// TwinCAT 3 PLC project PLC_PML
// ProgramVersion: 3.1.4023.0
// libraries:
//   Tc2_MC2, * (Beckhoff Automation GmbH)
//   Tc2_MC2_Drive, * (Beckhoff Automation GmbH)
//   Tc2_Standard, * (Beckhoff Automation GmbH)
//   Tc2_System, * (Beckhoff Automation GmbH)
//   Tc3_EventLogger, * (Beckhoff Automation GmbH)
//   Tc3_Module, * (Beckhoff Automation GmbH)
//   Tc3_PackML_V2, * (Beckhoff Automation GmbH)
// project tree:
//   Application/01_Application_Level_Items/02_DUT/01_ENUM/ E_PMLUnitMode.TcDUT
//   Application/01_Application_Level_Items/02_DUT/03_ALIAS/ T_PackMLTags.TcDUT
//   Application/01_Application_Level_Items/99_VISU/ V_Application.TcVIS
//   Application/02_MachineModules/ FB_TestMachine.TcPOU
//   Application/03_EquipmentModules/ FB_TestEquipment.TcPOU
//   Application/04_ControlModules/ FB_TestControl.TcPOU
//   Application/ MAIN.TcPOU
//   Base/01_PML/01_Module/01_Base/02_DUT/ ST_PMLModuleBase_HMI.TcDUT, ST_PMLModuleBase_VISU.TcDUT, ST_PMLSubUnitInfoExt.TcDUT
//   Base/01_PML/01_Module/01_Base/03_ITFs/ ITF_PMLModuleBase.TcIO
//   Base/01_PML/01_Module/01_Base/ FB_PMLModuleBase.TcPOU
//   Base/01_PML/01_Module/02_Events/ FB_PMLModeLogger.TcPOU, FB_PMLStateLogger.TcPOU
//   Base/01_PML/01_Module/03_PMLControl/03_ITFs/ ITF_PackML_ExternalControl.TcIO, ITF_PackML_ExternalControl_Simplified.TcIO
//   Base/01_PML/01_Module/03_PMLControl/ FB_ModuleExternalCommandControl.TcPOU, FB_PackML_ExternalControl.TcPOU, FB_PackML_PushButtonControl.TcPOU, ITF_PackML_ExternalControl_Simplified_old.TcIO
//   Base/01_PML/01_Module/04_SequenceControl/ E_ModuleSequenceCommand.TcDUT, E_ModuleSequenceStatus.TcDUT, F_CommandAllSequences.TcPOU, ITF_ModuleSequenceControl.TcIO, ST_ModuleSequenceControl.TcDUT
//   Base/01_PML/01_Module/05_Visualizations/ V_Module.TcVIS
//   Base/01_PML/02_GVL/ GVL_PML_Base.TcGVL
//   Base/01_PML/03_Visualizations/ V_MachineModule.TcVIS
//   Base/01_PML/99_Templates/01_ModuleTemplate/ FB_ApplicationModule_TEMPLATE.TcPOU
//   Base/02_Components/01_Base/ FB_ComponentBase.TcPOU, ITF_ComponentBase.TcIO, ST_ComponentBase_HMI.TcDUT
//   Base/02_Components/02_Axes/01_Base/ FB_AxisBase.TcPOU, ITF_AxisBase.TcIO, ST_AxisBase_HMI.TcDUT
//   Base/02_Components/02_Axes/02_Homing/ FB_Axis_HomeToSensor.TcPOU, FB_Axis_NoHoming.TcPOU
//   Base/02_Components/02_Axes/03_MotionType/ FB_Axis_Continuous_HomeToSensor.TcPOU, FB_Axis_Continuous_NoHoming.TcPOU, FB_Axis_Discrete_HomeToSensor.TcPOU, ITF_Axis_Continuous.TcIO, ITF_Axis_Discrete.TcIO
//   Base/02_Components/03_Cylinders/01_Base/ FB_CylinderBase.TcPOU, ITF_CylinderBase.TcIO, ST_CylinderBase_HMI.TcDUT
//   Base/02_Components/03_Cylinders/02_Feedback/ FB_Cylinder_DualSensor.TcPOU
//   Base/02_Components/03_Cylinders/03_Actuation/ FB_Cylinder_DualSolenoid_DualSensor.TcPOU
//   Base/02_Components/04_Sensors/01_Base/ E_DebounceMode.TcDUT, E_SensorSimulationMode.TcDUT, FB_SensorBase.TcPOU, ITF_SensorBase.TcIO, ST_SensorBase_HMI.TcDUT
//   Base/02_Components/04_Sensors/02_Sensor/ FB_Sensor.TcPOU
//   Base/03_Utilities/01_Events/ F_CreateAllEventsInClass.TcPOU
//   Base/03_Utilities/02_DataStructures/01_Tree/01_Tree_IndexBased/ FB_Tree_IndexBased.TcPOU, ITF_Tree_IndexBased.TcIO, ST_Tree_IndexBased_Node.TcDUT
//   Base/03_Utilities/03_HMI_Connections/ FB_MainHMI_Connection.TcPOU
//   / GlobalTextList.TcGTLO, PlcTask.TcTTO, Visualization Manager.TcVMO (not stored)
// real-time tasks:
//   TASK PlcTask: cycle T#1ms, priority 20, ADS port 350
//   TASK VISU_TASK: cycle T#200000us, priority 30, ADS port 351
//   TASK Job Task: cycle default, priority 32
//   TASK MC-Task (MET): cycle T#2ms, priority 3, ADS port 521
//   TASK MC-Task (MPT): cycle T#10ms, priority 8, ADS port 531
// motion (NC):
//   TASK NC-Task 1 SAF: cycle T#2ms, priority 4, ADS port 501
//   TASK NC-Task 1 SVB: cycle T#10ms, priority 9, ADS port 511
//   AXIS Axis 1 (id 1)
//     General: UnitFlags=#x00000004
//     Dynamic: AccelerationMaximum=10000, DecelerationMaximum=10000, Acceleration=1000, Deceleration=1000, Jerk=1750
//     Velo: Maximum=1500
//     OtherSettings: AllowMotionCmdToSlave=true
//     encoder EncType=1
//       EncPara: ModuloFactor=720
//     drive DrvType=5
//       Analog: TorqueSetpointScale=10, ScaleFactorActTorque=0.1
//       TimeComp: TaskDelayCycles=1
//     controller CtrType=1
//       CtrPara: PriorControlFactor=1
//         Observer: BandWidth=20
//   AXIS Axis 2 (id 2)
//     General: UnitFlags=#x00000004
//     OtherSettings: AllowMotionCmdToSlave=true
//     encoder EncType=1
//     drive DrvType=5
//       Analog: TorqueSetpointScale=10, ScaleFactorActTorque=0.1
//       TimeComp: TaskDelayCycles=1
//     controller CtrType=1
//       CtrPara: PriorControlFactor=1
//         Observer: BandWidth=20
// variable links:
//   PLC_PML/PLC_PML Instance <-> NC-Task 1 SAF/Axes/Axis 1
//     PlcTask Inputs/MAIN.fbMyMachine.fbEquipmentModule1.fb_EM1_ControlModule1.fbAxis1.HardwareAxis.NcToPlc <-> Outputs/ToPlc
//     PlcTask Outputs/MAIN.fbMyMachine.fbEquipmentModule1.fb_EM1_ControlModule1.fbAxis1.HardwareAxis.PlcToNc <-> Inputs/FromPlc
//   PLC_PML/PLC_PML Instance <-> NC-Task 1 SAF/Axes/Axis 2
//     PlcTask Inputs/MAIN.fbMyMachine.fbEquipmentModule1.fb_EM1_ControlModule1.fbAxis1.SimulationAxis.NcToPlc <-> Outputs/ToPlc
//     PlcTask Outputs/MAIN.fbMyMachine.fbEquipmentModule1.fb_EM1_ControlModule1.fbAxis1.SimulationAxis.PlcToNc <-> Inputs/FromPlc

CONFIGURATION PLC_PML
    RESOURCE PLC ON TwinCAT3
        TASK PlcTask(INTERVAL := T#1ms, PRIORITY := 20);
        PROGRAM MAIN WITH PlcTask : MAIN;
    END_RESOURCE
END_CONFIGURATION

// ---- Application/01_Application_Level_Items/02_DUT/01_ENUM/E_PMLUnitMode.TcDUT
{attribute 'qualified_only'}		//Note that this is not "Strict" since it needs to interact with the mode manager, which uses DINTs for mode
TYPE E_PMLUnitMode:
(
	ePMLUnitMode_Invalid 		:= 0,
	ePMLUnitMode_Production		:= 1,
	ePMLUnitMode_Maintenance	:= 2,
	ePMLUnitMode_Manual			:= 3
	// User defined modes
    (*ePMLUnitMode_SemiAutomatic  :=  4,
    ePMLUnitMode_DryRun         :=  5,
	ePMLUnitMode_Standalone		:=  6,
	ePMLUnitMode_Usermode4		:=  7,
	ePMLUnitMode_Usermode5 		:=  8,
	ePMLUnitMode_Usermode6 		:=  9,
	ePMLUnitMode_Usermode7 		:=  10 *)	
) DINT;
END_TYPE

// ---- Application/01_Application_Level_Items/02_DUT/03_ALIAS/T_PackMLTags.TcDUT
(*	Change the type depending on the needs, minimum packml set or full
Tc3_PackML_V2.ST_PackMLv30 // Tc3_PackML_V2.ST_PackMLv30min*)
TYPE T_PackMLTags : Tc3_PackML_V2.ST_PackMLv30; END_TYPE

// ---- Base/01_PML/01_Module/01_Base/02_DUT/ST_PMLModuleBase_HMI.TcDUT
TYPE ST_PMLModuleBase_HMI :
STRUCT
	bEnabled			: BOOL;					//Enables or disables the packml Machine of the module (prevents the module from going past idle)
	eMode				: E_PMLUnitMode;		//Current UnitMode of the module
	nModuleID			: DINT;					//Unique identifying number for the module
	sModuleName			: STRING;				//Human-readable module name for user-side messaging
	eState				: Tc3_PackML_V2.E_PMLState;
	bLogStateChanges 	: BOOL := TRUE; 		//Toggle to permit or suppress state change logging (Should be tied to HMI setting to optionally reduce event logger clutter)
	bLogModeChanges 	: BOOL := TRUE; 		//Toggle to permit or suppress state change logging (Should be tied to HMI setting to optionally reduce event logger clutter)
	
	//Control information
	bHMIControlAvailable	: BOOL;		//Set TRUE *FROM PLC* when HMI requests can be processed
	bIncomingHMIRequest 	: BOOL;		//Pulses TRUE when an HMI request is issued
	bHMICommandConfirmation	: BOOL;		//Confirms receipt and subsequent processing of the command sent by the HMI
	
	bModeCommandHMIRequest	: BOOL;		//Pulses TRUE when an HMI mode change request is issued
	bStateCommandHMIRequest	: BOOL;		//Pulses TRUE when an HMI state change request is issued
	bEnableHMIRequest				: BOOL;		//HMI requests to enable the module
	bDisableHMIRequest 				: BOOL;		//HMI requests to disable the module
	bActivateStateLogHMIRequest			: BOOL;		//HMI requests to enable the module
	bDeactivateStateLogHMIRequest 		: BOOL;		//HMI requests to disable the module
	bActivateModeLogHMIRequest			: BOOL;		//HMI requests to enable the module
	bDeactivateModeLogHMIRequest 		: BOOL;		//HMI requests to disable the module
	eModeCommandHMIValue			: E_PMLUnitMode;
	eStateCommandHMIValue			: Tc3_PackML_V2.E_PMLCommand;
	
END_STRUCT
END_TYPE

// ---- Base/01_PML/01_Module/01_Base/02_DUT/ST_PMLModuleBase_VISU.TcDUT
TYPE ST_PMLModuleBase_VISU :
STRUCT
	bEnabled			: BOOL;					//Enables or disables the packml Machine of the module (prevents the module from going past idle)
	eMode				: E_PMLUnitMode;		//Current UnitMode of the module
	nModuleID			: DINT;					//Unique identifying number for the module
	sModuleName			: STRING;				//Human-readable module name for user-side messaging
	eState				: Tc3_PackML_V2.E_PMLState;
	
	//eModeCommandValue	: E_PMLUnitMode;
	///eStateCommandValue	: Tc3_PackML_V2.E_PMLCommand;
	bStartPressed		: BOOL;
	///bStartEnabled		: BOOL;
	bStopPressed		: BOOL;
	///bStopEnabled		: BOOL;
	bResetPressed		: BOOL;
	///bResetEnabled		: BOOL;
	bClearPressed		: BOOL;
	///bClearEnabled		: BOOL;	
	
	bAbortPressed		: BOOL;
	bHoldPressed		: BOOL;
	bUnholdPressed		: BOOL;
	bSuspendPressed		: BOOL;
	bUnsuspendPressed	: BOOL;
	
	// Mode things
	bProductionPressed	: BOOL;
	bMaintenancePressed	: BOOL;
	bManualPressed		: BOOL;
	
END_STRUCT
END_TYPE

// ---- Base/01_PML/01_Module/01_Base/02_DUT/ST_PMLSubUnitInfoExt.TcDUT
TYPE ST_PMLSubUnitInfoExt EXTENDS ST_PMLSubUnitInfo :	//Extended Struct of ST_PMLSubUnitInfo
STRUCT
	nModuleID 						: DINT; 				//Machine ID for messaging and Identification
	sModuleName						: STRING;				//Human readable machine name for messaging
	UnitModeCurrent					: E_PMLProtectedUnitMode;
	ActiveAlarm						: BOOL;
END_STRUCT
END_TYPE

// ---- Base/01_PML/01_Module/04_SequenceControl/E_ModuleSequenceCommand.TcDUT
{attribute 'qualified_only'}
{attribute 'strict'}
TYPE E_ModuleSequenceCommand :
(
	Enable,
	Disable,
	Start,
	Resume,
	Reset,
	Clear	
);
END_TYPE

// ---- Base/01_PML/01_Module/04_SequenceControl/E_ModuleSequenceStatus.TcDUT
{attribute 'qualified_only'}
{attribute 'strict'}
TYPE E_ModuleSequenceStatus :
(
	Idle,
	Busy,
	Waiting,
	Complete,
	Disabled,
	Error
);
END_TYPE

// ---- Base/01_PML/01_Module/04_SequenceControl/ST_ModuleSequenceControl.TcDUT
TYPE ST_ModuleSequenceControl :
STRUCT
	eCommand				: E_ModuleSequenceCommand;	//Command Enumeration
	bNewCommand				: BOOL;						//Pulses TRUE when a new command is received
	bSequenceStateChange	: BOOL;						//TRUE when the sequence is transitioning between states, allows for one shot "on entry" tasks in sequence states 
	eStatus					: E_ModuleSequenceStatus;	//Abstracted and generalized status information for the local state machine status
END_STRUCT
END_TYPE

// ---- Base/02_Components/01_Base/ST_ComponentBase_HMI.TcDUT
TYPE ST_ComponentBase_HMI :
STRUCT
	//Status information
	bEnabled	: BOOL;
	bSimulate 	: BOOL;
	sName		: STRING;
	bActive		: BOOL;
	bError		: BOOL;
	nErrorID	: UDINT;
	
	//Control information
	bHMIControlAvailable	: BOOL;		//Set TRUE *FROM PLC* when HMI requests can be processed
	bIncomingHMIRequest 	: BOOL;		//Pulses TRUE when an HMI request is issued
	bHMICommandConfirmation	: BOOL;		//Confirms receipt and subsequent processing of the command sent by the HMI
	
	bEnableHMIRequest				: BOOL;		//HMI requests to enable the component
	bDisableHMIRequest 				: BOOL;		//HMI requests to disable the component
	bSimulateOperationHMIRequest 	: BOOL;		//HMI requests to change the component to simulation mode
	bStandardOperationHMIRequest	: BOOL;		//HMI requests to change the component to standard mode
	bResetHMIRequest				: BOOL;		//HMI requests to reset the component
	
END_STRUCT
END_TYPE

// ---- Base/02_Components/02_Axes/01_Base/ST_AxisBase_HMI.TcDUT
TYPE ST_AxisBase_HMI :
STRUCT
	fJogFastVelocity	: LREAL;
	fJogSlowVelocity	: LREAL;
	fTargetVelocity		: LREAL;
	
	bDriveEnabled		: BOOL;
	bInGear				: BOOL;
	bInPosition			: BOOL;
	fPosition 			: LREAL;
	fPositionSetpoint	: LREAL;
	bStopped			: BOOL;
	
	//Control information
	bHMIControlAvailable	: BOOL;		//Set TRUE *FROM PLC* when HMI requests can be processed
	bIncomingHMIRequest 	: BOOL;		//Pulses TRUE when an HMI request is issued
		bHMICommandConfirmation	: BOOL;		//Confirms receipt and subsequent processing of the command sent by the HMI
	
	bDriveEnableHMIRequest				: BOOL;		//HMI requests to enable the axis
	bDriveDisableHMIRequest 				: BOOL;		//HMI requests to disable the axis
	bSetJogFastVelocityRequest		: BOOL;
	bSetJogSlowVelocityRequest		: BOOL;
	fSetJogFastVelocityValue		: LREAL;
	fSetJogSlowVelocityValue		: LREAL;
	bSetTargetVelocityRequest		: BOOL;
	bSetTargetVelocityValue			: LREAL;
END_STRUCT
END_TYPE

// ---- Base/02_Components/03_Cylinders/01_Base/ST_CylinderBase_HMI.TcDUT
TYPE ST_CylinderBase_HMI:
STRUCT
	//Status information
	tExtendTime		: TIME;
	tRetractTime	: TIME;
	fTimeoutFactor	: LREAL;
	bExtended		: BOOL;
	bRetracted		: BOOL;
	bExtending		: BOOL;
	bRetracting		: BOOL;
	bRetractCommand	: BOOL;
	bExtendCommand	: BOOL;
	
	//Control information
	bHMIControlAvailable	: BOOL;		//Set TRUE *FROM PLC* when HMI requests can be processed
	bIncomingHMIRequest 	: BOOL;		//Pulses TRUE when an HMI request is issued
		bHMICommandConfirmation	: BOOL;		//Confirms receipt and subsequent processing of the command sent by the HMI
	
	bExtendHMIRequest			: BOOL;			//HMI requests to extend the cylinder
	bRetractHMIRequest			: BOOL;			//HMI requests to retract the cylinder
	bIdleHMIRequest				: BOOL;			//HMI requests to idle the cylinder (no active output)
	bExtendTimeHMISetRequest	: BOOL;			//HMI requests to set the cylinder's expected extend time
	tExtendTimeHMISetValue		: TIME;			//HMI setpoint value for the expected extend time
	bRetractTimeHMISetRequest	: BOOL;			//HMI requests to set the cylinder's expected retract time
	tRetractTimeHMISetValue		: TIME;			//HMI setpoint value for the expected retract time
	bTimeoutFactorHMISetRequest	: BOOL;			//HMI requests to set the timeout factor for the cylinder
	fTimeoutFactorHMISetValue	: LREAL;		//HMI setpoint value for the cylinder's timeout factor
END_STRUCT
END_TYPE

// ---- Base/02_Components/04_Sensors/01_Base/E_DebounceMode.TcDUT
{attribute 'qualified_only'}
{attribute 'strict'}
TYPE E_DebounceMode :
(
	RawInput,
	SimpleFlickerFilter,
	EdgeDetectFilter,
	MovingAverage
) DINT;
END_TYPE

// ---- Base/02_Components/04_Sensors/01_Base/E_SensorSimulationMode.TcDUT
{attribute 'qualified_only'}
{attribute 'strict'}
TYPE E_SensorSimulationMode :
(
	InputDriven,		//Follows the state of the SimulationInput property
	Periodic			//Follows a 50% duty cycle at the period specified in ms by SimulationInput);
);
END_TYPE

// ---- Base/02_Components/04_Sensors/01_Base/ST_SensorBase_HMI.TcDUT
TYPE ST_SensorBase_HMI :
STRUCT
	//Status information
	eDebounceMode		: E_DebounceMode;
	tDebounceTime 		: TIME;
	bInverted			: BOOL;
	eSimulationMode		: E_SensorSimulationMode;
	nSimulationInput	: DINT;
	tTimeActive			: TIME;
	tTimeInactive		: TIME;
	
	//Control information
	bHMIControlAvailable	: BOOL;		//Set TRUE *FROM PLC* when HMI requests can be processed
	bIncomingHMIRequest 	: BOOL;		//Pulses TRUE when an HMI request is issued
		bHMICommandConfirmation	: BOOL;		//Confirms receipt and subsequent processing of the command sent by the HMI
	
	bSetDebounceModeHMIRequest 		: BOOL;		//HMI requests to change the Debounce mode of the sensor
	eSetDebounceModeHMIValue 		: E_DebounceMode;			//HMI requested Debounce mode of the sensor
	bSetDebounceTimeHMIRequest		: BOOL;		//HMI requests to change the Debounce time of the sensor
	tSetDebounceTimeHMIValue 		: TIME;	//HMI requested Debounce mode of the sensor
	bSetSimulationModeHMIRequest	: BOOL;		//HMI requests to change the simulation mode of the sensor
	eSetSimulationModeHMIValue		: E_SensorSimulationMode;	//HMI Requested Simulation mode of the sensor
	bSetSimulationInputHMIRequest	: BOOL;		//HMI requests to set the simulation input value
	nSetSimulationInputHMIValue		: DINT;		//HMI requested simulation input value
	bInvertedHMIRequest				: BOOL;		//HMI requests that the sensor operate in an inverted state
	bUninvertedHMIRequest			: BOOL;		//HMI requests that the sensor operate in an uninverted state
	
	bSimulateOperationHMIRequest 	: BOOL;		//HMI requests to change the component to simulation mode
	bStandardOperationHMIRequest	: BOOL;		//HMI requests to change the component to standard mode

END_STRUCT
END_TYPE

// ---- Base/03_Utilities/02_DataStructures/01_Tree/01_Tree_IndexBased/ST_Tree_IndexBased_Node.TcDUT
TYPE ST_Tree_IndexBased_Node :
STRUCT
	sName 		: STRING;
	nChildCount	: DINT;
	nParent		: DINT;
	a_nChildren	: ARRAY[0..15] OF DINT;
	nDepth		: DINT;
END_STRUCT
END_TYPE

// ---- Base/01_PML/02_GVL/GVL_PML_Base.TcGVL
///{attribute 'qualified_only'}
VAR_GLOBAL



	nAxis: INT;
END_VAR

VAR_GLOBAL CONSTANT
	MAX_NO_OF_SUBUNITS			: UDINT := 20;

	ePMLUNITMODEDEFAULT			: E_PMLUnitMode := E_PMLUnitMode.ePMLUnitMode_Production;
	ePMLSTATEDEFAULT			: E_PMLCommand := E_PMLCommand.ePMLCommand_Abort;

END_VAR

// ---- Base/01_PML/01_Module/01_Base/03_ITFs/ITF_PMLModuleBase.TcIO
INTERFACE ITF_PMLModuleBase EXTENDS ITF_UnitState

PROPERTY AncestorIDs : STRING
GET
END_GET
SET
END_SET
END_PROPERTY

METHOD CyclicLogic
VAR_INPUT
END_VAR
END_METHOD

PROPERTY Enabled : BOOL
GET
END_GET
SET
END_SET
END_PROPERTY

PROPERTY LogModeChanges : BOOL
GET
END_GET
SET
END_SET
END_PROPERTY

PROPERTY LogStateChanges : BOOL
GET
END_GET
SET
END_SET
END_PROPERTY

PROPERTY Mode : E_PMLUnitMode
GET
END_GET
END_PROPERTY

PROPERTY ModeCommand : DINT
SET
END_SET
END_PROPERTY

PROPERTY ModuleID : DINT
GET
END_GET
SET
END_SET
END_PROPERTY

PROPERTY ModuleName : STRING
GET
END_GET
SET
END_SET
END_PROPERTY

PROPERTY State : E_PMLState
GET
END_GET
END_PROPERTY

PROPERTY StateCommand : E_PMLCommand
SET
END_SET
END_PROPERTY

END_INTERFACE

// ---- Base/01_PML/01_Module/03_PMLControl/03_ITFs/ITF_PackML_ExternalControl.TcIO
INTERFACE ITF_PackML_ExternalControl EXTENDS ITF_PackML_ExternalControl_Simplified

PROPERTY Mode : DINT
GET
END_GET
SET
END_SET
END_PROPERTY

PROPERTY ModeCommand : DINT
GET
END_GET
SET
END_SET
END_PROPERTY

PROPERTY ModeCommandPulse : BOOL
GET
END_GET
SET
END_SET
END_PROPERTY

PROPERTY State : E_PMLState
GET
END_GET
SET
END_SET
END_PROPERTY

PROPERTY StateCommand : E_PMLCommand
GET
END_GET
SET
END_SET
END_PROPERTY

PROPERTY StateCommandPulse : BOOL
GET
END_GET
SET
END_SET
END_PROPERTY

END_INTERFACE

// ---- Base/01_PML/01_Module/03_PMLControl/03_ITFs/ITF_PackML_ExternalControl_Simplified.TcIO
INTERFACE ITF_PackML_ExternalControl_Simplified

{warning 'add property implementation'}
PROPERTY ClearEnabled : BOOL
GET
END_GET
SET
END_SET
END_PROPERTY

{warning 'add property implementation'}
PROPERTY ClearPressed : BOOL
GET
END_GET
SET
END_SET
END_PROPERTY

PROPERTY ResetEnabled : BOOL
GET
END_GET
SET
END_SET
END_PROPERTY

PROPERTY ResetPressed : BOOL
GET
END_GET
SET
END_SET
END_PROPERTY

PROPERTY StartEnabled : BOOL
GET
END_GET
SET
END_SET
END_PROPERTY

PROPERTY StartPressed : BOOL
GET
END_GET
SET
END_SET
END_PROPERTY

PROPERTY StopEnabled : BOOL
GET
END_GET
SET
END_SET
END_PROPERTY

PROPERTY StopPressed : BOOL
GET
END_GET
SET
END_SET
END_PROPERTY

END_INTERFACE

// ---- Base/01_PML/01_Module/03_PMLControl/ITF_PackML_ExternalControl_Simplified_old.TcIO
INTERFACE ITF_PackML_ExternalControl_Simplified_old

PROPERTY ClearEnabled : BOOL
GET
END_GET
SET
END_SET
END_PROPERTY

PROPERTY ClearPressed : BOOL
GET
END_GET
SET
END_SET
END_PROPERTY

PROPERTY ResetEnabled : BOOL
GET
END_GET
SET
END_SET
END_PROPERTY

PROPERTY ResetPressed : BOOL
GET
END_GET
SET
END_SET
END_PROPERTY

PROPERTY StartEnabled : BOOL
GET
END_GET
SET
END_SET
END_PROPERTY

PROPERTY StartPressed : BOOL
GET
END_GET
SET
END_SET
END_PROPERTY

PROPERTY StopEnabled : BOOL
GET
END_GET
SET
END_SET
END_PROPERTY

PROPERTY StopPressed : BOOL
GET
END_GET
SET
END_SET
END_PROPERTY

END_INTERFACE

// ---- Base/01_PML/01_Module/04_SequenceControl/ITF_ModuleSequenceControl.TcIO
INTERFACE ITF_ModuleSequenceControl

METHOD ClearSequence : BOOL
VAR_INPUT
END_VAR
END_METHOD

METHOD DisableSequence : BOOL
END_METHOD

METHOD EnableSequence : BOOL
END_METHOD

METHOD ResetSequence : BOOL
END_METHOD

METHOD ResumeSequence : BOOL
VAR_INPUT
END_VAR
END_METHOD

PROPERTY SequenceCommand : E_ModuleSequenceCommand
GET
END_GET
SET
END_SET
END_PROPERTY

PROPERTY SequenceStatus : E_ModuleSequenceStatus
GET
END_GET
END_PROPERTY

METHOD StartSequence : BOOL
END_METHOD

END_INTERFACE

// ---- Base/02_Components/01_Base/ITF_ComponentBase.TcIO
INTERFACE ITF_ComponentBase

PROPERTY Active : BOOL	//TRUE when the component is in motion or otherwise completing a commanded task
GET
END_GET
END_PROPERTY

METHOD CyclicLogic : BOOL		//Should be called Externally akin to the PML Modules
END_METHOD

PROPERTY Enabled : BOOL	//Enables or disables the component
GET
END_GET
SET
END_SET
END_PROPERTY

PROPERTY Error : BOOL	//Boolean to signal that an error has ocurred
GET
END_GET
END_PROPERTY

PROPERTY ErrorID : UDINT	//Integer ID to identify the proper alarm to be posted from the parent module
GET
END_GET
SET
END_SET
END_PROPERTY

PROPERTY Name : STRING
GET
END_GET
SET
END_SET
END_PROPERTY

METHOD Reset : BOOL
END_METHOD

{warning 'add property implementation'}
PROPERTY Simulate : BOOL
GET
END_GET
SET
END_SET
END_PROPERTY

END_INTERFACE

// ---- Base/02_Components/02_Axes/01_Base/ITF_AxisBase.TcIO
INTERFACE ITF_AxisBase

PROPERTY AxisRef : AXIS_REF
GET
END_GET
END_PROPERTY

PROPERTY DriveEnabled : BOOL
GET
END_GET
END_PROPERTY

METHOD GearInBasic : BOOL
VAR_IN_OUT
	master : AXIS_REF;	//Master axis to which the gearing will be made
END_VAR
END_METHOD

METHOD Home : BOOL
END_METHOD

PROPERTY InGear : BOOL
GET
END_GET
END_PROPERTY

METHOD Inhibit : BOOL
VAR_INPUT
END_VAR
END_METHOD

PROPERTY InPosition : BOOL
GET
END_GET
END_PROPERTY

METHOD Jog : BOOL
VAR_INPUT
	direction	: BOOL;			//"TRUE" for positive jog, "FALSE" for negative jog
	fast		: BOOL;			//"TRUE" for 'fast' jog, "FALSE" for 'slow' jog (As defined by Jog(Slow/Fast)Velocity Property)
END_VAR
END_METHOD

PROPERTY JogFastVelocity : LREAL
GET
END_GET
SET
END_SET
END_PROPERTY

PROPERTY JogSlowVelocity : LREAL
GET
END_GET
SET
END_SET
END_PROPERTY

METHOD MovePosition : BOOL
VAR_INPUT
	override 	: BOOL := FALSE;		//Allows this instruction to override another ongoing operation(This parameter is initialized so that once default parameter value functionality is added to TwinCAT, this input will not need to be set explicitly in the Method call)
	position	: LREAL;				//Desired position to which the axis should move
END_VAR
END_METHOD

METHOD MoveRelative : BOOL
VAR_INPUT
	override 	: BOOL := FALSE;		//Allows this instruction to override another ongoing operation(This parameter is initialized so that once default parameter value functionality is added to TwinCAT, this input will not need to be set explicitly in the Method call)
	distance 	: LREAL;				//Desired distance to be moved
END_VAR
END_METHOD

METHOD MoveVelocity : BOOL
VAR_INPUT
	override	: BOOL := FALSE;				//Allows this instruction to override another ongoing operation(This parameter is initialized so that once default parameter value functionality is added to TwinCAT, this input will not need to be set explicitly in the Method call)
	velocity	: LREAL;		//Desired velocity for the axis
END_VAR
END_METHOD

PROPERTY Position : LREAL
GET
END_GET
END_PROPERTY

PROPERTY PositionSetpoint : LREAL
GET
END_GET
END_PROPERTY

METHOD Stop : BOOL
END_METHOD

PROPERTY Stopped : BOOL
GET
END_GET
END_PROPERTY

PROPERTY TargetVelocity : LREAL
GET
END_GET
SET
END_SET
END_PROPERTY

METHOD Uninhibit : BOOL
VAR_INPUT
END_VAR
END_METHOD

END_INTERFACE

// ---- Base/02_Components/02_Axes/03_MotionType/ITF_Axis_Continuous.TcIO
INTERFACE ITF_Axis_Continuous

PROPERTY ModuloFactor : LREAL
GET
END_GET
END_PROPERTY

PROPERTY ModuloPosition : LREAL
GET
END_GET
END_PROPERTY

METHOD SetAxisModuloFactor : BOOL
VAR_INPUT
	fSetAxisModuloFactor		: LREAL;
END_VAR
END_METHOD

END_INTERFACE

// ---- Base/02_Components/02_Axes/03_MotionType/ITF_Axis_Discrete.TcIO
INTERFACE ITF_Axis_Discrete

PROPERTY LowerTravelLimit : LREAL
GET
END_GET
SET
END_SET
END_PROPERTY

PROPERTY Position_1 : LREAL
GET
END_GET
SET
END_SET
END_PROPERTY

PROPERTY Position_2 : LREAL
GET
END_GET
SET
END_SET
END_PROPERTY

PROPERTY Position_3 : LREAL
GET
END_GET
SET
END_SET
END_PROPERTY

PROPERTY UpperTravelLimit : LREAL
GET
END_GET
SET
END_SET
END_PROPERTY

END_INTERFACE

// ---- Base/02_Components/03_Cylinders/01_Base/ITF_CylinderBase.TcIO
INTERFACE ITF_CylinderBase//cylinder no feedback spring return solonoid

METHOD Extend : BOOL
END_METHOD

PROPERTY Extended : BOOL	//Status bit for the position of the cylinder
GET
END_GET
END_PROPERTY

PROPERTY Extending : BOOL
GET
END_GET
END_PROPERTY

PROPERTY ExtendTime : TIME	//Approximate expected time for the cylinder to complete an extension cycle
GET
END_GET
SET
END_SET
END_PROPERTY

METHOD Idle : BOOL
END_METHOD

METHOD Retract : UDINT
END_METHOD

PROPERTY Retracted : BOOL	//Status bit for the position of the cylinder
GET
END_GET
END_PROPERTY

PROPERTY Retracting : BOOL
GET
END_GET
END_PROPERTY

PROPERTY RetractTime : TIME
GET
END_GET
SET
END_SET
END_PROPERTY

PROPERTY TimeoutFactor : LREAL	//Multiplicative factor that determines error timeout threshold based on the expected time
GET
END_GET
SET
END_SET
END_PROPERTY

END_INTERFACE

// ---- Base/02_Components/04_Sensors/01_Base/ITF_SensorBase.TcIO
INTERFACE ITF_SensorBase

PROPERTY DebounceMode : E_DebounceMode
GET
END_GET
SET
END_SET
END_PROPERTY

PROPERTY DebounceTime : TIME
GET
END_GET
SET
END_SET
END_PROPERTY

PROPERTY Inverted : BOOL		//"High" signal from the sensor will be interpreted as an "inactive" reading when this parameter is TRUE
GET
END_GET
SET
END_SET
END_PROPERTY

PROPERTY SimulationInput : DINT
GET
END_GET
SET
END_SET
END_PROPERTY

PROPERTY SimulationMode : E_SensorSimulationMode
GET
END_GET
SET
END_SET
END_PROPERTY

PROPERTY TimeActive : TIME
GET
END_GET
END_PROPERTY

PROPERTY TimeInactive : TIME
GET
END_GET
END_PROPERTY

END_INTERFACE

// ---- Base/03_Utilities/02_DataStructures/01_Tree/01_Tree_IndexBased/ITF_Tree_IndexBased.TcIO
INTERFACE ITF_Tree_IndexBased

METHOD AddNodeAsChildByName : BOOL
VAR_INPUT
	sNewName 	: STRING;
	sParentName	: STRING;
END_VAR
END_METHOD

END_INTERFACE

// ---- Application/MAIN.TcPOU
PROGRAM MAIN
VAR
	// Define the top level Machine as defined in the Application/01_MachineModules folder here
	fbMyMachine				: FB_TestMachine;	
	fbMainHMIConnection		: FB_MainHMI_Connection;

	bInitialized			: BOOL;
END_VAR

CyclicLogic();

METHOD CyclicLogic : BOOL
VAR_INPUT
END_VAR
IF NOT bInitialized THEN
	Initialize();
	bInitialized := TRUE;
END_IF

//The Top level machine CyclicLogic call should be made here, all sub modules should be called from within their respective parent CyclicLogic methods
fbMyMachine.CyclicLogic();


// Add other Main CyclicLogic here
fbMainHMIConnection();
END_METHOD

METHOD Initialize : BOOL
VAR_INPUT
END_VAR
//Top level machine initialization should happen here, in the main initialization method. Each subsequent "layer" of modules will be named within their respective "parent" intialize method
fbMainHMIConnection.sTopLevelMachine := fbMyMachine.ModuleName;

fbMyMachine.iMasterDataStructure_Adder 	:= fbMainHMIConnection.DataStructure_Adder;
fbMyMachine.Enabled 					:=  TRUE;
fbMyMachine.ModuleName 					:=  'Test Machine';
fbMyMachine.ModuleID 					:=  1;
fbMyMachine.AncestorIDs 				:= '';

fbMainHMIConnection(sTopLevelMachine 	:= fbMyMachine.ModuleName);
END_METHOD

END_PROGRAM

// ---- Application/02_MachineModules/FB_TestMachine.TcPOU
FUNCTION_BLOCK FB_TestMachine EXTENDS FB_PMLModuleBase
VAR
	//Define the Sub modules here for this module.  Also set the Interfaces in the initialize method.
	//fbSubModule1				: FB_ApplicationModule_TEMPLATE;		// Sub module instantiation
	//fbSubModule2				: FB_ApplicationModule_TEMPLATE;		// Sub module instantiation
	
	fbEquipmentModule1			: FB_TestEquipment;
	
	//temporary array of module base interfaces to be copied over to the base class itfPackMLBase variable
	a_itfPackMLBase_init		: ARRAY[1..MAX_NO_OF_SUBUNITS] OF ITF_PMLModuleBase := [fbEquipmentModule1](*, fbSubModule2,*);

	// Other machine specific variables here
END_VAR

//*********************************************************
// Code implementation only in Execute() method for consistency with templates
//*********************************************************

// 
// Cyclic Code
METHOD CyclicLogic
VAR
	i								: UDINT;		//Generic iteration value
END_VAR
// Main loop of the parent module
SUPER^.CyclicLogic();
END_METHOD

METHOD Initialize
VAR
	i								: UDINT;		//Generic iteration value
END_VAR

// Define the interfaces to the different subunits (Must take place before SUPER^.initialize call)
FOR i := 1 TO MAX_NO_OF_SUBUNITS DO
	a_itfPackMLBase[i] := a_itfPackMLBase_init[i];
END_FOR

fbEquipmentModule1.iMasterDataStructure_Adder 	:= iMasterDataStructure_Adder;
fbEquipmentModule1.Enabled 						:=  TRUE;
fbEquipmentModule1.ModuleName 					:=  'Test Equipment 1';
fbEquipmentModule1.ModuleID 					:=  1;
fbEquipmentModule1.AncestorIDs 					:= CONCAT(CONCAT(sAncestorIDs, DINT_TO_STRING(nModuleID)), '_');

iMasterDataStructure_Adder.AddNodeAsChildByName(fbEquipmentModule1.ModuleName, sModuleName);

// Init of the parent class object (Must be called AFTER most local init code, since the sub module interface array assignments should be made here, and then operated on within the module base init
SUPER^.Initialize();
END_METHOD

END_FUNCTION_BLOCK

// ---- Base/01_PML/01_Module/01_Base/FB_PMLModuleBase.TcPOU
FUNCTION_BLOCK ABSTRACT FB_PMLModuleBase IMPLEMENTS ITF_PMLModuleBase, ITF_UnitState, ITF_ModuleSequenceControl
VAR_INPUT
	iMasterDataStructure_Adder		: ITF_Tree_IndexBased;			//Interface for adding new children to the master machine tree data representation
END_VAR
VAR
	//ITF_PackMLBase internal property variables
	bEnabled			: BOOL;					//Enables or disables the packml Machine of the module (prevents the module from going past idle)
	eMode				: E_PMLUnitMode;		//Current UnitMode of the module
	eModeCommand		: E_PMLUnitMode; 				//Current Commanded UnitMode of the module
	nModuleID			: DINT;					//Unique identifying number for the module
	sModuleName			: STRING;				//Human-readable module name for user-side messaging
	eState				: Tc3_PackML_V2.E_PMLState;
	eStateCommand		: Tc3_PackML_V2.E_PMLCommand;
	bLogStateChanges 	: BOOL := TRUE; 		//Toggle to permit or suppress state change logging (Should be tied to HMI setting to optionally reduce event logger clutter)
	bLogModeChanges 	: BOOL := TRUE; 		//Toggle to permit or suppress state change logging (Should be tied to HMI setting to optionally reduce event logger clutter)

	stPMLModuleBaseHMI	: ST_PMLModuleBase_HMI;		//Handles atatus and cointrol communications with the HMI
	stPMLModuleBaseVISU	: ST_PMLModuleBase_VISU;	//Handles the status and control with Visulizations

	//Administration of FB Variables
	bInitialized 					: BOOL;					//TRUE when initialization code of the object is complete
	sAncestorIDs					: STRING;				//String concatenation of preceding parent IDs to prefix this module's ID
	sID_Name						: STRING;				//"Module XX - 'Module Name' " Alarm and message utility phrase based off of nMachine ID and sMachineName
	fbExternalControl				: FB_ModuleExternalCommandControl;
	// Packtags data
	//{attribute 'OPC.UA.DA' := '1'}
	//{attribute 'OPC.UA.DA.StructuredType' := '1'}
	//packTags						: T_PackMLTags;		//PackTags instantiation
	
	//State and Mode control
	fbModeManager 					: PML_UnitModeManager; 	//Manages operating mode transitions and rules
	fbStateMachine 					: PML_StateMachine; 	//Manages PackML state transitions
	fbCustomModes 					: PML_UnitModeConfig;	//Used to define custom machine modes if desired

	//State and Mode Status and Command variables
	sState							: STRING; 				//String representation of the current state
	eLastState						: E_PMLState;			//Last cycle PackML state
	eLastStateCommand				: E_PMLCommand;			//Previous received PackML state command
	eLastMode		 				: DINT;					//Last PackML mode 
	eLastModeCommand 				: E_PMLUnitMode;					//Previous received PackML mode command
	bStateTasksComplete				: BOOL;					//All tasks to be performed at this program level are complete
	bSubModulesReady				: BOOL;					//All submodules have reached the commanded state
	
	//Alarming and Logging variables - Some may or may not be necessary depending on final alarm system implementation ----------------------------------------------
	//These are for the newer TMC Excel import style alarm system
	a_fbPMLAlarms						: ARRAY[1..48] OF FB_TcAlarm;	//Array of alarms for PackML state and mode changes that exist in any PackML enabled module
	a_fbBaseAlarms					: ARRAY[1..32] OF FB_TcAlarm;		//Array of alarms for general module Alarms				
	fbPMLStateLogger				: FB_PMLStateLogger;	//Logs PackML state changes
	fbPMLModeLogger					: FB_PMLModeLogger;	//Logs PackML Mode changes

	// Alarm handling
	bActiveAlarm					: BOOL;					//module has an active alarm					

	//Sequence Control Structure
	stSequenceControl 		: ST_ModuleSequenceControl;		//Provides variables with which the ModuleSequenceControl interface may interact 

	//********************************************************************************************************************
	// Sub Module variables
	// Used mostly for EMs and Machines, but ok for CM. They are just null	
	a_itfPackMLBase					: ARRAY[1..MAX_NO_OF_SUBUNITS] OF ITF_PMLModuleBase;
	// Array of the PML sub unit info array used by the statemachine
	a_stPMLSubUnitInfo				: ARRAY[1..MAX_NO_OF_SUBUNITS] OF ST_PMLSubUnitInfo;
	udNumberOfSubUnits				: UDINT := 0;	//Defined number of instantiated Module
	// This is the information for each modules subunits.
	PMLSubUnitInfoRef				: ST_PMLSubUnitInfoRef;				// Reference to the subunit information, used by the state machine
	//********************************************************************************************************************
	
END_VAR

//*********************************************************
// !!!!! Code implementation only in CyclicLogic() method !!!!! 
//*********************************************************

PROPERTY AncestorIDs : STRING
GET
AncestorIDs := sAncestorIDs;
END_GET
SET
sAncestorIDs := AncestorIDs;
END_SET
END_PROPERTY

METHOD ClearSequence : BOOL
VAR_INPUT
END_VAR
stSequenceControl.eCommand := E_ModuleSequenceCommand.Clear;
stSequenceControl.bNewCommand := TRUE;
END_METHOD

METHOD CreateEvents : BOOL
VAR_INPUT
END_VAR

VAR
	bCreated1: BOOL;
	bCreated2: BOOL;
END_VAR

bCreated1 := F_CreateAllEventsInClass(	p_aAlarms := a_fbPMLAlarms,
							nClassSize := SIZEOF(TC_EVENTS.PMLAlarms),
							pInitEvent := ADR(TC_EVENTS.PMLAlarms.InitReferenceEvent),
							sPrefix := sID_Name);
							
bCreated2 := F_CreateAllEventsInClass(	p_aAlarms := a_fbBaseAlarms,
							nClassSize := SIZEOF(TC_EVENTS.BaseAlarms),
							pInitEvent := ADR(TC_EVENTS.BaseAlarms.InitReferenceEvent),
							sPrefix := sID_Name);
END_METHOD

// 
// Cyclic Code
METHOD CyclicLogic


VAR
	i: UDINT;
END_VAR
//*********************************************************
//If you are about to write actual machine implementation code, note that implementation code should exist within an implementation machine module block that extends this machine module base!
//*********************************************************

// First loop initialization code is triggered by highest level class
IF NOT bInitialized THEN			//Force initialization code of the object
	initialize();
	bInitialized := TRUE;
END_IF

//  call the subunits
FOR i := 1 TO udNumberOfSubUnits DO
	a_itfPackMLBase[i].CyclicLogic();								//Call the main cyclic loop of the subunits 
	a_stPMLSubUnitInfo[i].eState := a_itfPackMLBase[i].State;  	//Reflect the state of the subunits to the state machine of the module
END_FOR

// Mode control loop of the module
M_ModeControl();

// State control loop of the module
M_StateControl();

HMICommunication();
VISUCommunication();
fbExternalControl();
END_METHOD

METHOD DisableSequence : BOOL
stSequenceControl.eCommand := E_ModuleSequenceCommand.Disable;
stSequenceControl.bNewCommand := TRUE;
END_METHOD

PROPERTY Enabled : BOOL
GET
Enabled := bEnabled;
END_GET
SET
bEnabled := Enabled;
END_SET
END_PROPERTY

METHOD EnableSequence : BOOL
stSequenceControl.eCommand := E_ModuleSequenceCommand.Enable;
stSequenceControl.bNewCommand := TRUE;
END_METHOD

METHOD HMICommunication : BOOL
//Extend this method in extended FBs to communicate specific implementation data

//Process HMI requests
IF stPMLModuleBaseHMI.bIncomingHMIRequest AND NOT stPMLModuleBaseHMI.bHMICommandConfirmation THEN		//If a request has been issued by the HMI, and a previous request has not just finished being processed
	IF stPMLModuleBaseHMI.bHMIControlAvailable THEN		//If the current conditions permit HMI control (Should be determined by the extended application components)
		IF stPMLModuleBaseHMI.bEnableHMIRequest THEN
			bEnabled := TRUE;
			stPMLModuleBaseHMI.bHMICommandConfirmation := TRUE;	//Confirm that the request has been processed
		END_IF
		IF stPMLModuleBaseHMI.bDisableHMIRequest THEN
			bEnabled := FALSE;
			stPMLModuleBaseHMI.bHMICommandConfirmation := TRUE;	//Confirm that the request has been processed
		END_IF
		IF stPMLModuleBaseHMI.bModeCommandHMIRequest THEN
			//KAB eModeCommand := stPMLModuleBaseHMI.eModeCommandHMIValue;
			fbExternalControl.ExternalControlHMI.ModeCommand := stPMLModuleBaseHMI.eModeCommandHMIValue;
			stPMLModuleBaseHMI.bHMICommandConfirmation := TRUE;	//Confirm that the request has been processed
		END_IF
		IF stPMLModuleBaseHMI.bStateCommandHMIRequest THEN
			//KAB eStateCommand := stPMLModuleBaseHMI.eStateCommandHMIValue;
			fbExternalControl.ExternalControlHMI.StateCommand := stPMLModuleBaseHMI.eStateCommandHMIValue;
			stPMLModuleBaseHMI.bHMICommandConfirmation := TRUE;	//Confirm that the request has been processed
		END_IF
	END_IF
	
		//The following commands are always permissible, and are therefore not conditioned with bHMIControlAvailable
	IF stPMLModuleBaseHMI.bActivateStateLogHMIRequest THEN
		bLogStateChanges := TRUE;
		stPMLModuleBaseHMI.bHMICommandConfirmation := TRUE;	//Confirm that the request has been processed
	END_IF
	IF stPMLModuleBaseHMI.bDeactivateStateLogHMIRequest THEN
		bLogStateChanges := FALSE;
		stPMLModuleBaseHMI.bHMICommandConfirmation := TRUE;	//Confirm that the request has been processed
	END_IF
	IF stPMLModuleBaseHMI.bActivateModeLogHMIRequest THEN
		bLogModeChanges := TRUE;
		stPMLModuleBaseHMI.bHMICommandConfirmation := TRUE;	//Confirm that the request has been processed
	END_IF
	IF stPMLModuleBaseHMI.bDeactivateModeLogHMIRequest THEN
		bLogModeChanges := FALSE;
		stPMLModuleBaseHMI.bHMICommandConfirmation := TRUE;	//Confirm that the request has been processed
	END_IF		
END_IF


//Update HMI status info
stPMLModuleBaseHMI.bEnabled := bEnabled;
stPMLModuleBaseHMI.eMode := fbExternalControl.ExternalControlHMI.Mode;		//KAB eMode;
stPMLModuleBaseHMI.nModuleID := nModuleID;
stPMLModuleBaseHMI.sModuleName := sModuleName;
stPMLModuleBaseHMI.eState := fbExternalControl.ExternalControlHMI.State;	//KAB eState;
stPMLModuleBaseHMI.bLogStateChanges := bLogStateChanges;
stPMLModuleBaseHMI.bLogModeChanges := bLogModeChanges;
END_METHOD

METHOD initialize
VAR
	i : UDINT;
END_VAR
sID_Name := CONCAT(CONCAT(CONCAT(CONCAT(CONCAT('Module ', sAncestorIDs), DINT_TO_STRING(nModuleID)), ' - '), sModuleName), ' '); 	//Creates a utility string for alarms and other messaging that reads (example text) - "Module 10 - Main Casepacker" to be followed by the alarm or message info

// Figure out how many SubUnits - they should be from 1 to X and not skip any.
udNumberOfSubUnits := 0;
FOR i:=1 TO MAX_NO_OF_SUBUNITS DO
	IF a_itfPackMLBase[i] <> 0 THEN
		udNumberOfSubUnits:=udNumberOfSubUnits+1;
	END_IF
END_FOR

fbExternalControl.Module := THIS^;

// <BASIC INITIALIZATION CODE, DO NOT CHANGE>
// Initialize subunit overview used by state machine
PMLSubUnitInfoRef.ArraySize := SIZEOF(a_stPMLSubUnitInfo);
PMLSubUnitInfoRef.NoOfSubUnits := udNumberOfSubUnits;
PMLSubUnitInfoRef.pArray := ADR(a_stPMLSubUnitInfo);
// Point the state machine to the locally defined subunit info 
fbStateMachine.stSubUnitInfoRef := PMLSubUnitInfoRef;
// <\BASIC INITIALIZATION CODE, DO NOT CHANGE>

// Activate all subunits by default, or change accordingly
FOR i:=1 TO udNumberOfSubUnits DO
	a_stPMLSubUnitInfo[i].Active	:= TRUE;					// Follows Main State Machine
END_FOR

CreateEvents();
END_METHOD

PROPERTY LogModeChanges : BOOL
GET
LogModeChanges:= bLogModeChanges;
END_GET
SET
bLogModeChanges := LogModeChanges;
END_SET
END_PROPERTY

PROPERTY LogStateChanges : BOOL
GET
LogStateChanges:= bLogStateChanges;
END_GET
SET
bLogStateChanges := LogStateChanges;
END_SET
END_PROPERTY

METHOD M_Aborted
//*************************************************************************************************************************************************************************
//If you are about to write application specific code, note that any such code should exist within the "Application" directory using a Function Block that 'EXTENDS' this base Function Block!
//This particular method's functionality can be overriden in the extended block by creating a method of the same name, with desired functionality therein
//If the functionality of this base module is to be retained, but more functionality is desired, the extended method can contain a SUPER^.ThisMethodName(); call, which will call this code
//*************************************************************************************************************************************************************************

;
END_METHOD

{attribute 'object_name' := 'M_Aborting'}
METHOD M_Aborting
VAR
	nModuleNo							: UDINT;		//Generic iteration value
END_VAR
//*************************************************************************************************************************************************************************
//If you are about to write application specific code, note that any such code should exist within the "Application" directory using a Function Block that 'EXTENDS' this base Function Block!
//This particular method's functionality can be overriden in the extended block by creating a method of the same name, with desired functionality therein
//If the functionality of this base module is to be retained, but more functionality is desired, the extended method can contain a SUPER^.ThisMethodName(); call, which will call this code
//*************************************************************************************************************************************************************************

//Perform State tasks here
// Send abort command to all sub modules
FOR nModuleNo := 1 TO udNumberOfSubUnits DO
	a_itfPackMLBase[nModuleNo].StateCommand:=ePMLCommand_Abort;
END_FOR

bStateTasksComplete := TRUE;		//Sending the command is all that is necessary by default, if more functionality is needed at this level, add it above and condition this value appropriately

// All subunits in requested state?
bSubModulesReady := TRUE;
FOR nModuleNo := 1 TO udNumberOfSubUnits DO
	bSubModulesReady := bSubModulesReady AND (a_itfPackMLBase[nModuleNo].State = ePMLState_Aborted);
END_FOR
IF bSubModulesReady AND bStateTasksComplete THEN
	bStateTasksComplete := FALSE;
	M_StateComplete();
END_IF
END_METHOD

{attribute 'object_name' := 'M_Clearing'}
METHOD M_Clearing
VAR
	nModuleNo							: UDINT;		//Generic iteration value
END_VAR
//*************************************************************************************************************************************************************************
//If you are about to write application specific code, note that any such code should exist within the "Application" directory using a Function Block that 'EXTENDS' this base Function Block!
//This particular method's functionality can be overriden in the extended block by creating a method of the same name, with desired functionality therein
//If the functionality of this base module is to be retained, but more functionality is desired, the extended method can contain a SUPER^.ThisMethodName(); call, which will call this code
//*************************************************************************************************************************************************************************

//Perform State tasks here
// Send clear command to all sub modules
FOR nModuleNo := 1 TO udNumberOfSubUnits DO	
	a_itfPackMLBase[nModuleNo].StateCommand	:=	ePMLCommand_Clear;
END_FOR

bStateTasksComplete := TRUE;		//Sending the command is all that is necessary by default, if more functionality is needed at this level, add it above and condition this value appropriately

// All subunits in requested state?
bSubModulesReady	:= TRUE;
FOR nModuleNo := 1 TO udNumberOfSubUnits DO
	bSubModulesReady := bSubModulesReady AND (a_itfPackMLBase[nModuleNo].State = ePMLState_Stopped);
END_FOR
IF bSubModulesReady AND bStateTasksComplete THEN
	bStateTasksComplete := FALSE;
	M_StateComplete();
END_IF
END_METHOD

METHOD M_Complete
//*************************************************************************************************************************************************************************
//If you are about to write application specific code, note that any such code should exist within the "Application" directory using a Function Block that 'EXTENDS' this base Function Block!
//This particular method's functionality can be overriden in the extended block by creating a method of the same name, with desired functionality therein
//If the functionality of this base module is to be retained, but more functionality is desired, the extended method can contain a SUPER^.ThisMethodName(); call, which will call this code
//*************************************************************************************************************************************************************************

;
END_METHOD

{attribute 'object_name' := 'M_Completing'}
METHOD M_Completing
VAR
	nModuleNo							: UDINT;		//Generic iteration value
END_VAR
//*************************************************************************************************************************************************************************
//If you are about to write application specific code, note that any such code should exist within the "Application" directory using a Function Block that 'EXTENDS' this base Function Block!
//This particular method's functionality can be overriden in the extended block by creating a method of the same name, with desired functionality therein
//If the functionality of this base module is to be retained, but more functionality is desired, the extended method can contain a SUPER^.ThisMethodName(); call, which will call this code
//*************************************************************************************************************************************************************************

//Perform State tasks here
// Send complete command to all sub modules
FOR nModuleNo := 1 TO udNumberOfSubUnits DO
	a_itfPackMLBase[nModuleNo].StateCommand:=ePMLCommand_Complete;
END_FOR

bStateTasksComplete := TRUE;		//Sending the command is all that is necessary by default, if more functionality is needed at this level, add it above and condition this value appropriately

// All subunits in requested state?
bSubModulesReady	:= TRUE;
FOR nModuleNo := 1 TO udNumberOfSubUnits DO
	bSubModulesReady := bSubModulesReady AND (a_itfPackMLBase[nModuleNo].State = ePMLState_Complete);
END_FOR
IF bSubModulesReady AND bStateTasksComplete THEN
	bStateTasksComplete := FALSE;
	M_StateComplete();
END_IF
END_METHOD

METHOD M_Execute
//*************************************************************************************************************************************************************************
//If you are about to write application specific code, note that any such code should exist within the "Application" directory using a Function Block that 'EXTENDS' this base Function Block!
//This particular method's functionality can be overriden in the extended block by creating a method of the same name, with desired functionality therein
//If the functionality of this base module is to be retained, but more functionality is desired, the extended method can contain a SUPER^.ThisMethodName(); call, which will call this code
//*************************************************************************************************************************************************************************

;
END_METHOD

METHOD M_Held
//*************************************************************************************************************************************************************************
//If you are about to write application specific code, note that any such code should exist within the "Application" directory using a Function Block that 'EXTENDS' this base Function Block!
//This particular method's functionality can be overriden in the extended block by creating a method of the same name, with desired functionality therein
//If the functionality of this base module is to be retained, but more functionality is desired, the extended method can contain a SUPER^.ThisMethodName(); call, which will call this code
//*************************************************************************************************************************************************************************
END_METHOD

{attribute 'object_name' := 'M_Holding'}
METHOD M_Holding
VAR
	nModuleNo							: UDINT;		//Generic iteration value
END_VAR
//*************************************************************************************************************************************************************************
//If you are about to write application specific code, note that any such code should exist within the "Application" directory using a Function Block that 'EXTENDS' this base Function Block!
//This particular method's functionality can be overriden in the extended block by creating a method of the same name, with desired functionality therein
//If the functionality of this base module is to be retained, but more functionality is desired, the extended method can contain a SUPER^.ThisMethodName(); call, which will call this code
//*************************************************************************************************************************************************************************

//Perform State tasks here
// Send hold command to all sub modules
FOR nModuleNo := 1 TO udNumberOfSubUnits DO
	a_itfPackMLBase[nModuleNo].StateCommand:=ePMLCommand_Hold;
END_FOR

bStateTasksComplete := TRUE;		//Sending the command is all that is necessary by default, if more functionality is needed at this level, add it above and condition this value appropriately

// All subunits in requested state?
bSubModulesReady	:= TRUE;
FOR nModuleNo := 1 TO udNumberOfSubUnits DO
	bSubModulesReady := bSubModulesReady AND (a_itfPackMLBase[nModuleNo].State = ePMLState_Held);
END_FOR
IF bSubModulesReady AND bStateTasksComplete THEN
	bStateTasksComplete := FALSE;
	M_StateComplete();
END_IF
END_METHOD

METHOD M_Idle
//*************************************************************************************************************************************************************************
//If you are about to write application specific code, note that any such code should exist within the "Application" directory using a Function Block that 'EXTENDS' this base Function Block!
//This particular method's functionality can be overriden in the extended block by creating a method of the same name, with desired functionality therein
//If the functionality of this base module is to be retained, but more functionality is desired, the extended method can contain a SUPER^.ThisMethodName(); call, which will call this code
//*************************************************************************************************************************************************************************
END_METHOD

METHOD PRIVATE M_ModeControl
VAR
	i					: UDINT;
END_VAR
//On startup, Mode is invalid, set it to production
IF eMode = E_PMLUnitMode.ePMLUnitMode_Invalid 		THEN 
	fbModeManager.bExecute 		:= TRUE; 
	eModeCommand			 	:= ePMLUNITMODEDEFAULT; 
	eLastModeCommand 			:= eModeCommand;
//If mode is valid and the command has changed, attempt to change modes
ELSIF eModeCommand <> eLastModeCommand 					THEN
	//DONKEY : logging to be implemented
	fbModeManager.bExecute 		:= TRUE;
	eLastModeCommand 			:= eModeCommand;
END_IF

//Handles mode changes based on eModeCommand and the state transition rules defined in the pre-defined protected modes or custom modes
fbModeManager(
	eModeCommand			:= eModeCommand, 
	eState					:= eState, 			
	eModeStatus				=> eMode, 
	bDone					=> , 
	bError					=> , 
	nErrorId				=> 
	);

// Reset mode control command
eModeCommand := E_PMLUnitMode.ePMLUnitMode_Invalid;
fbModeManager.bExecute 		:= FALSE;

//If PackML mode has changed
IF fbModeManager.eModeStatus <> eLastMode  THEN 
	eLastMode := fbModeManager.eModeStatus; 
	//If state change logging is not suppressed
 	IF bLogStateChanges THEN 
		fbPMLModeLogger(
			a_fbPMLAlarms := a_fbPMLAlarms,
			sModulePrefix := sID_Name,
			Mode := fbModeManager.eModeStatus);	
	END_IF	
	// Change SubModules
	FOR i := 1 TO udNumberOfSubUnits DO
		a_itfPackMLBase[i].ModeCommand := fbModeManager.eModeStatus;		//Call the SetMode loop of the subunits 
	END_FOR

END_IF
END_METHOD

{attribute 'object_name' := 'M_Resetting'}
METHOD M_Resetting
VAR
	nModuleNo							: UDINT;		//Generic iteration value
END_VAR
//*************************************************************************************************************************************************************************
//If you are about to write application specific code, note that any such code should exist within the "Application" directory using a Function Block that 'EXTENDS' this base Function Block!
//This particular method's functionality can be overriden in the extended block by creating a method of the same name, with desired functionality therein
//If the functionality of this base module is to be retained, but more functionality is desired, the extended method can contain a SUPER^.ThisMethodName(); call, which will call this code
//*************************************************************************************************************************************************************************

//Perform State tasks here
// Send clear/reset command to all sub modules
//As long as this module is in the "Resetting" state, it will attempt to get all modules to Idle by sending abort, clear, and reset commands as appropriate to its children until they do
FOR nModuleNo := 1 TO udNumberOfSubUnits DO
	IF a_itfPackMLBase[nModuleNo].State=ePMLState_Stopped THEN
		a_itfPackMLBase[nModuleNo].StateCommand:=ePMLCommand_Reset;
	ELSIF a_itfPackMLBase[nModuleNo].State=ePMLState_Aborted THEN
		a_itfPackMLBase[nModuleNo].StateCommand:=ePMLCommand_Clear;
	ELSIF a_itfPackMLBase[nModuleNo].State=ePMLState_Clearing OR a_itfPackMLBase[nModuleNo].State=ePMLState_Stopping 
		OR a_itfPackMLBase[nModuleNo].State=ePMLState_Resetting OR a_itfPackMLBase[nModuleNo].State=ePMLState_Idle THEN
		;
	ELSE
		a_itfPackMLBase[nModuleNo].StateCommand:=ePMLCommand_Abort;
	END_IF
END_FOR

bStateTasksComplete := TRUE;		//Sending the command is all that is necessary by default, if more functionality is needed at this level, add it above and condition this value appropriately

// All subunits in requested state?
bSubModulesReady	:= TRUE;
FOR nModuleNo := 1 TO udNumberOfSubUnits DO
	bSubModulesReady := bSubModulesReady AND (a_itfPackMLBase[nModuleNo].State = ePMLState_Idle);
END_FOR
IF bSubModulesReady AND bStateTasksComplete THEN
	bStateTasksComplete := FALSE;
	M_StateComplete();
END_IF
END_METHOD

{attribute 'object_name' := 'M_Starting'}
METHOD M_Starting
VAR
	nModuleNo							: UDINT;		//Generic iteration value
END_VAR
//*************************************************************************************************************************************************************************
//If you are about to write application specific code, note that any such code should exist within the "Application" directory using a Function Block that 'EXTENDS' this base Function Block!
//This particular method's functionality can be overriden in the extended block by creating a method of the same name, with desired functionality therein
//If the functionality of this base module is to be retained, but more functionality is desired, the extended method can contain a SUPER^.ThisMethodName(); call, which will call this code
//*************************************************************************************************************************************************************************

//Perform State tasks here
// Send start command to all sub modules
FOR nModuleNo := 1 TO udNumberOfSubUnits DO
	a_itfPackMLBase[nModuleNo].StateCommand:=ePMLCommand_Start;
END_FOR

bStateTasksComplete := TRUE;		//Sending the command is all that is necessary by default, if more functionality is needed at this level, add it above and condition this value appropriately

// All subunits in requested state?
bSubModulesReady	:= TRUE;
FOR nModuleNo := 1 TO udNumberOfSubUnits DO
	bSubModulesReady := bSubModulesReady AND (a_itfPackMLBase[nModuleNo].State = ePMLState_Execute);
END_FOR
IF bSubModulesReady AND bStateTasksComplete THEN
	bStateTasksComplete := FALSE;
	M_StateComplete();
END_IF
END_METHOD

METHOD M_StateComplete
//*************************************************************************************************************************************************************************
//If you are about to write application specific code, note that any such code should exist within the "Application" directory using a Function Block that 'EXTENDS' this base Function Block!
//This particular method's functionality can be overriden in the extended block by creating a method of the same name, with desired functionality therein
//If the functionality of this base module is to be retained, but more functionality is desired, the extended method can contain a SUPER^.ThisMethodName(); call, which will call this code
//*************************************************************************************************************************************************************************

fbStateMachine.M_StateComplete();
END_METHOD

METHOD PRIVATE M_StateControl
//On startup, state is invalid, set it to default
IF eState = E_PMLState.ePMLState_Undefined 				AND 
	eMode <> E_PMLUnitMode.ePMLUnitMode_Invalid 	THEN 
	eStateCommand 	:= ePMLSTATEDEFAULT; 
END_IF

//If mode is valid and the command has changed, attempt to change modes
IF eStateCommand <> eLastModeCommand 							AND 
	eMode <> E_PMLUnitMode.ePMLUnitMode_Invalid 	THEN
	IF bLogStateChanges THEN 
		//DONKEY : logging to be implemented
		//Simple string insertion, if event class based implementation is desired, follow FB_PMLStateLogger as a template for FB_PMLCommandLogger
		//Logger.logMessage(msg:= CONCAT(ConCAT(deviceIDMessage,' PLC Requests  '), F_CommandStateToString(eStateCommand)));   
		;
	END_IF		
	eLastStateCommand 			:= eStateCommand;
END_IF

//Call PackML state machine	
fbStateMachine(
	eMode				:= eMode, 
	eCommand			:= eStateCommand, 
	stSubUnitInfoRef	:= ,
	stOptions			:= , 
	eState				=> eState, 
	sState 				=> sState, 
	bError				=> , 
	nErrorID			=> );

//If PackML state has changed
IF eState <> eLastState  THEN 
	eLastState := eState; 
	//If state change logging is not suppressed
 	IF bLogStateChanges THEN 
		fbPMLStateLogger(
			a_fbPMLAlarms := a_fbPMLAlarms, 
			sModulePrefix := SID_Name, 
			eState := eState);	
	END_IF	
END_IF 
	
//*********************************************************
//If you are about to write actual machine implementation code, note that implementation code should exist within an implementation equipment module block that extends this equipment module base!
//*********************************************************

// Call appropriate method depending on current PackML state
CASE eState OF
	E_PMLState.ePMLState_Undefined:
		M_Undefined();
	E_PMLState.ePMLState_Clearing:
		M_Clearing();
	E_PMLState.ePMLState_Stopped:
		M_Stopped();
	E_PMLState.ePMLState_Starting:
		M_Starting();
	E_PMLState.ePMLState_Idle:
		M_Idle();
	E_PMLState.ePMLState_Suspended:
		M_Suspended();
	E_PMLState.ePMLState_Execute:
		M_Execute();
	E_PMLState.ePMLState_Stopping:
		M_Stopping();
	E_PMLState.ePMLState_Aborting:
		M_Aborting();
	E_PMLState.ePMLState_Aborted:
		M_Aborted();
	E_PMLState.ePMLState_Holding:
		M_Holding();
	E_PMLState.ePMLState_Held:
		M_Held();
	E_PMLState.ePMLState_Unholding:
		M_Unholding();
	E_PMLState.ePMLState_Suspending:
		M_Suspending();
	E_PMLState.ePMLState_Unsuspending:
		M_Unsuspending();
	E_PMLState.ePMLState_Resetting:   	
		M_Resetting();
	E_PMLState.ePMLState_Completing:
		M_Completing();
	E_PMLState.ePMLState_Complete:
		M_Complete();
END_CASE
END_METHOD

METHOD M_Stopped
//*************************************************************************************************************************************************************************
//If you are about to write application specific code, note that any such code should exist within the "Application" directory using a Function Block that 'EXTENDS' this base Function Block!
//This particular method's functionality can be overriden in the extended block by creating a method of the same name, with desired functionality therein
//If the functionality of this base module is to be retained, but more functionality is desired, the extended method can contain a SUPER^.ThisMethodName(); call, which will call this code
//*************************************************************************************************************************************************************************
END_METHOD

{attribute 'object_name' := 'M_Stopping'}
METHOD M_Stopping
VAR
	nModuleNo							: UDINT;		//Generic iteration value
END_VAR
//*************************************************************************************************************************************************************************
//If you are about to write application specific code, note that any such code should exist within the "Application" directory using a Function Block that 'EXTENDS' this base Function Block!
//This particular method's functionality can be overriden in the extended block by creating a method of the same name, with desired functionality therein
//If the functionality of this base module is to be retained, but more functionality is desired, the extended method can contain a SUPER^.ThisMethodName(); call, which will call this code
//*************************************************************************************************************************************************************************

//Perform State tasks here
// Send stop command to all sub modules
FOR nModuleNo := 1 TO udNumberOfSubUnits DO
	a_itfPackMLBase[nModuleNo].StateCommand:=ePMLCommand_Stop;
END_FOR

bStateTasksComplete := TRUE;		//Sending the command is all that is necessary by default, if more functionality is needed at this level, add it above and condition this value appropriately

// All subunits in requested state?
bSubModulesReady	:= TRUE;
FOR nModuleNo := 1 TO udNumberOfSubUnits DO
	bSubModulesReady := bSubModulesReady AND (a_itfPackMLBase[nModuleNo].State = ePMLState_Stopped);
END_FOR
IF bSubModulesReady AND bStateTasksComplete THEN
	bStateTasksComplete := FALSE;
	M_StateComplete();
END_IF
END_METHOD

METHOD M_Suspended
//*************************************************************************************************************************************************************************
//If you are about to write application specific code, note that any such code should exist within the "Application" directory using a Function Block that 'EXTENDS' this base Function Block!
//This particular method's functionality can be overriden in the extended block by creating a method of the same name, with desired functionality therein
//If the functionality of this base module is to be retained, but more functionality is desired, the extended method can contain a SUPER^.ThisMethodName(); call, which will call this code
//*************************************************************************************************************************************************************************
END_METHOD

{attribute 'object_name' := 'M_Suspending'}
METHOD M_Suspending
VAR
	nModuleNo							: UDINT;		//Generic iteration value
END_VAR
//*************************************************************************************************************************************************************************
//If you are about to write application specific code, note that any such code should exist within the "Application" directory using a Function Block that 'EXTENDS' this base Function Block!
//This particular method's functionality can be overriden in the extended block by creating a method of the same name, with desired functionality therein
//If the functionality of this base module is to be retained, but more functionality is desired, the extended method can contain a SUPER^.ThisMethodName(); call, which will call this code
//*************************************************************************************************************************************************************************

//Perform State tasks here
// Send suspend command to all sub modules
FOR nModuleNo := 1 TO udNumberOfSubUnits DO
	a_itfPackMLBase[nModuleNo].StateCommand:=ePMLCommand_Suspend;
END_FOR

bStateTasksComplete := TRUE;		//Sending the command is all that is necessary by default, if more functionality is needed at this level, add it above and condition this value appropriately

// All subunits in requested state?
bSubModulesReady	:= TRUE;
FOR nModuleNo := 1 TO udNumberOfSubUnits DO
	bSubModulesReady := bSubModulesReady AND (a_itfPackMLBase[nModuleNo].State = ePMLState_Suspended);
END_FOR
IF bSubModulesReady AND bStateTasksComplete THEN
	bStateTasksComplete := FALSE;
	M_StateComplete();
END_IF
END_METHOD

METHOD M_Undefined
//*************************************************************************************************************************************************************************
//If you are about to write application specific code, note that any such code should exist within the "Application" directory using a Function Block that 'EXTENDS' this base Function Block!
//This particular method's functionality can be overriden in the extended block by creating a method of the same name, with desired functionality therein
//If the functionality of this base module is to be retained, but more functionality is desired, the extended method can contain a SUPER^.ThisMethodName(); call, which will call this code
//*************************************************************************************************************************************************************************
END_METHOD

{attribute 'object_name' := 'M_Unholding'}
METHOD M_Unholding
VAR
	nModuleNo							: UDINT;		//Generic iteration value
END_VAR
//*************************************************************************************************************************************************************************
//If you are about to write application specific code, note that any such code should exist within the "Application" directory using a Function Block that 'EXTENDS' this base Function Block!
//This particular method's functionality can be overriden in the extended block by creating a method of the same name, with desired functionality therein
//If the functionality of this base module is to be retained, but more functionality is desired, the extended method can contain a SUPER^.ThisMethodName(); call, which will call this code
//*************************************************************************************************************************************************************************

//Perform State tasks here
// Send unhold command to all sub modules
FOR nModuleNo := 1 TO udNumberOfSubUnits DO
	a_itfPackMLBase[nModuleNo].StateCommand:=ePMLCommand_Unhold;
END_FOR

bStateTasksComplete := TRUE;		//Sending the command is all that is necessary by default, if more functionality is needed at this level, add it above and condition this value appropriately

// All subunits in requested state?
bSubModulesReady	:= TRUE;
FOR nModuleNo := 1 TO udNumberOfSubUnits DO
	bSubModulesReady := bSubModulesReady AND (a_itfPackMLBase[nModuleNo].State = ePMLState_Execute);
END_FOR
IF bSubModulesReady AND bStateTasksComplete THEN
	bStateTasksComplete := FALSE;
	M_StateComplete();
END_IF
END_METHOD

{attribute 'object_name' := 'M_Unsuspending'}
METHOD M_Unsuspending
VAR
	nModuleNo							: UDINT;		//Generic iteration value
END_VAR
//*************************************************************************************************************************************************************************
//If you are about to write application specific code, note that any such code should exist within the "Application" directory using a Function Block that 'EXTENDS' this base Function Block!
//This particular method's functionality can be overriden in the extended block by creating a method of the same name, with desired functionality therein
//If the functionality of this base module is to be retained, but more functionality is desired, the extended method can contain a SUPER^.ThisMethodName(); call, which will call this code
//*************************************************************************************************************************************************************************

//Perform State tasks here
// Send unsuspend command to all sub modules
FOR nModuleNo := 1 TO udNumberOfSubUnits DO
	a_itfPackMLBase[nModuleNo].StateCommand:=ePMLCommand_Unsuspend;
END_FOR

bStateTasksComplete := TRUE;		//Sending the command is all that is necessary by default, if more functionality is needed at this level, add it above and condition this value appropriately

// All subunits in requested state?
bSubModulesReady	:= TRUE;
FOR nModuleNo := 1 TO udNumberOfSubUnits DO
	bSubModulesReady := bSubModulesReady AND (a_itfPackMLBase[nModuleNo].State = ePMLState_Execute);
END_FOR
IF bSubModulesReady AND bStateTasksComplete THEN
	bStateTasksComplete := FALSE;
	M_StateComplete();
END_IF
END_METHOD

PROPERTY Mode : E_PMLUnitMode
GET
Mode := eMode;
END_GET
END_PROPERTY

PROPERTY ModeCommand : DINT
SET
eModeCommand := ModeCommand;
END_SET
END_PROPERTY

PROPERTY ModuleID : DINT
GET
ModuleID := nModuleID;
END_GET
SET
nModuleID := ModuleID;
END_SET
END_PROPERTY

PROPERTY ModuleName : STRING
GET
ModuleName := sModuleName;
END_GET
SET
sModuleName := ModuleName;
END_SET
END_PROPERTY

METHOD ResetSequence : BOOL
stSequenceControl.eCommand := E_ModuleSequenceCommand.Reset;
stSequenceControl.bNewCommand := TRUE;
END_METHOD

METHOD ResumeSequence : BOOL
VAR_INPUT
END_VAR
stSequenceControl.eCommand := E_ModuleSequenceCommand.Resume;
stSequenceControl.bNewCommand := TRUE;
END_METHOD

PROPERTY SequenceCommand : E_ModuleSequenceCommand
GET
SequenceCommand := stSequenceControl.eCommand;
END_GET
SET
stSequenceControl.eCommand := SequenceCommand;
END_SET
END_PROPERTY

PROPERTY SequenceStatus : E_ModuleSequenceStatus
GET
SequenceStatus := stSequenceControl.eStatus;
END_GET
END_PROPERTY

METHOD StartSequence : BOOL
stSequenceControl.eCommand := E_ModuleSequenceCommand.Start;
stSequenceControl.bNewCommand := TRUE;
END_METHOD

PROPERTY State : Tc3_PackML_V2.E_PMLState
GET
State := eState;
END_GET
END_PROPERTY

PROPERTY StateCommand : Tc3_PackML_V2.E_PMLCommand
SET
IF 	eMode <> E_PMLUnitMode.ePMLUnitMode_Invalid 	AND
 	eState <> E_PMLState.ePMLState_Undefined 			THEN 
	eStateCommand := StateCommand;
END_IF
END_SET
END_PROPERTY

METHOD VISUCommunication : BOOL
VAR_INPUT
END_VAR

fbExternalControl.ExternalControlVISU.ClearPressed := stPMLModuleBaseVISU.bClearPressed;
fbExternalControl.ExternalControlVISU.ResetPressed := stPMLModuleBaseVISU.bResetPressed;
fbExternalControl.ExternalControlVISU.StartPressed := stPMLModuleBaseVISU.bStartPressed;
fbExternalControl.ExternalControlVISU.StopPressed := stPMLModuleBaseVISU.bStopPressed;


//Update VISU status info
stPMLModuleBaseVISU.bEnabled := bEnabled;
stPMLModuleBaseVISU.eMode := eMode;		
stPMLModuleBaseVISU.nModuleID := nModuleID;
stPMLModuleBaseVISU.sModuleName := sModuleName;
stPMLModuleBaseVISU.eState := eState;	

// Mode logic here.  Only taking the button from the visualizations
IF stPMLModuleBaseVISU.bProductionPressed AND eMode <> E_PMLUnitMode.ePMLUnitMode_Production THEN
	fbExternalControl.ExternalControlVISU.ModeCommand := E_PMLUnitMode.ePMLUnitMode_Production;
	fbExternalControl.ExternalControlVISU.ModeCommandPulse := TRUE;
END_IF
IF stPMLModuleBaseVISU.bMaintenancePressed AND eMode <> E_PMLUnitMode.ePMLUnitMode_Maintenance THEN
	fbExternalControl.ExternalControlVISU.ModeCommand := E_PMLUnitMode.ePMLUnitMode_Maintenance;
	fbExternalControl.ExternalControlVISU.ModeCommandPulse := TRUE;
END_IF
IF stPMLModuleBaseVISU.bManualPressed AND eMode <> E_PMLUnitMode.ePMLUnitMode_Manual THEN
	fbExternalControl.ExternalControlVISU.ModeCommand := E_PMLUnitMode.ePMLUnitMode_Manual;
	fbExternalControl.ExternalControlVISU.ModeCommandPulse := TRUE;
END_IF

// Extra buttons from Visu here for state changes than the standard 4
// Abort
IF stPMLModuleBaseVISU.bAbortPressed THEN
	CASE eState OF
		ePMLState_Aborted,
		ePMLState_Aborting:
			// DO Nothing
	ELSE
		fbExternalControl.ExternalControlVISU.StateCommand := E_PMLCommand.ePMLCommand_Abort;
		fbExternalControl.ExternalControlVISU.StateCommandPulse := TRUE;	
	END_CASE
END_IF

// Hold
IF stPMLModuleBaseVISU.bHoldPressed THEN
	IF eState = ePMLState_Execute THEN
		fbExternalControl.ExternalControlVISU.StateCommand := E_PMLCommand.ePMLCommand_Hold;
		fbExternalControl.ExternalControlVISU.StateCommandPulse := TRUE;	
	END_IF
END_IF

// unHold
IF stPMLModuleBaseVISU.bUnholdPressed THEN
	IF eState = ePMLState_Held THEN
		fbExternalControl.ExternalControlVISU.StateCommand := E_PMLCommand.ePMLCommand_Unhold;
		fbExternalControl.ExternalControlVISU.StateCommandPulse := TRUE;	
	END_IF
END_IF

// Suspend
IF stPMLModuleBaseVISU.bSuspendPressed THEN
	IF eState = ePMLState_Execute THEN
		fbExternalControl.ExternalControlVISU.StateCommand := E_PMLCommand.ePMLCommand_Suspend;
		fbExternalControl.ExternalControlVISU.StateCommandPulse := TRUE;	
	END_IF
END_IF

// unSuspend
IF stPMLModuleBaseVISU.bUnsuspendPressed THEN
	IF eState = ePMLState_Suspended THEN
		fbExternalControl.ExternalControlVISU.StateCommand := E_PMLCommand.ePMLCommand_Unsuspend;
		fbExternalControl.ExternalControlVISU.StateCommandPulse := TRUE;	
	END_IF
END_IF
END_METHOD

END_FUNCTION_BLOCK

// ---- Base/01_PML/01_Module/03_PMLControl/FB_ModuleExternalCommandControl.TcPOU
FUNCTION_BLOCK FB_ModuleExternalCommandControl
VAR_INPUT
END_VAR
VAR_OUTPUT
END_VAR
VAR
	ipModulePackMLBase		: ITF_PMLModuleBase;
	
	fbHMIControl				: FB_PackML_ExternalControl;
	fbVISUControl				: FB_PackML_ExternalControl;
	fbPushButtonControl			: FB_PackML_PushButtonControl;
			
	a_iExternalControlSources	: ARRAY[1..3] OF ITF_PackML_ExternalControl := [fbHMIControl,fbVISUControl,fbPushButtonControl];	//Add more control sources as desired
	
	i : DINT;
END_VAR

FOR i := 1 TO 3 DO		//TODO: Make Dynamic through constant declaration or otherwise
	
	IF a_iExternalControlSources[i].ModeCommandPulse THEN
		ipModulePackMLBase.ModeCommand := a_iExternalControlSources[i].ModeCommand;
		a_iExternalControlSources[i].ModeCommandPulse := FALSE;
	END_IF
	
	IF a_iExternalControlSources[i].StateCommandPulse THEN
		ipModulePackMLBase.StateCommand := a_iExternalControlSources[i].StateCommand;
		a_iExternalControlSources[i].StateCommandPulse := FALSE;
	END_IF
	
	a_iExternalControlSources[i].Mode := ipModulePackMLBase.Mode;
	a_iExternalControlSources[i].State := ipModulePackMLBase.State;
END_FOR

fbHMIControl();
fbVISUControl();
///fbPushButtonControl();

PROPERTY ExternalControlHMI : ITF_PackML_ExternalControl
GET
ExternalControlHMI := a_iExternalControlSources[1];
END_GET
END_PROPERTY

PROPERTY ExternalControlVISU : ITF_PackML_ExternalControl
GET
ExternalControlVISU := a_iExternalControlSources[2];
END_GET
END_PROPERTY

PROPERTY Module : ITF_PMLModuleBase
GET
Module := ipModulePackMLBase;
END_GET
SET
ipModulePackMLBase := Module;
END_SET
END_PROPERTY

END_FUNCTION_BLOCK

// ---- Base/01_PML/01_Module/03_PMLControl/FB_PackML_ExternalControl.TcPOU
FUNCTION_BLOCK FB_PackML_ExternalControl IMPLEMENTS ITF_PackML_ExternalControl
VAR_INPUT
END_VAR
VAR_OUTPUT
END_VAR
VAR
	nMode				: DINT;
	nModeCommand		: DINT;
	bModeCommandPulse	: BOOL;
	eState				: Tc3_PackML_V2.E_PMLState;
	eStateCommand		: Tc3_PackML_V2.E_PMLCommand;
	bStateCommandPulse	: BOOL;
	
	bStartPressed		: BOOL;
	bStartEnabled		: BOOL;
	bStopPressed		: BOOL;
	bStopEnabled		: BOOL;
	bResetPressed		: BOOL;
	bResetEnabled		: BOOL;
	bClearPressed		: BOOL;
	bClearEnabled		: BOOL;	
	
END_VAR

//Handle button presses
IF bStartPressed THEN
	IF eState = Tc3_PackML_V2.E_PMLState.ePMLState_Idle THEN
		eStateCommand := Tc3_PackML_V2.E_PMLCommand.ePMLCommand_Start;
		bStateCommandPulse := TRUE;
	ELSIF eState = Tc3_PackML_V2.E_PMLState.ePMLState_Held THEN
		eStateCommand := Tc3_PackML_V2.E_PMLCommand.ePMLCommand_Unhold;
		bStateCommandPulse := TRUE;
	END_IF
	bStartPressed := FALSE;
END_IF

IF bStopPressed THEN
	eStateCommand := Tc3_PackML_V2.E_PMLCommand.ePMLCommand_Stop;
	bStateCommandPulse := TRUE;
	bStopPressed := FALSE;
END_IF

IF bResetPressed THEN
	eStateCommand := Tc3_PackML_V2.E_PMLCommand.ePMLCommand_Reset;
	bStateCommandPulse := TRUE;
	bResetPressed := FALSE;
END_IF

IF bClearPressed THEN
	eStateCommand := Tc3_PackML_V2.E_PMLCommand.ePMLCommand_Clear;
	bStateCommandPulse := TRUE;
	bClearPressed := FALSE;
END_IF

//Handle enabling of the Start button
IF 		eState = Tc3_PackML_V2.E_PMLState.ePMLState_Idle
	OR	eState = Tc3_PackML_V2.E_PMLState.ePMLState_Held 	THEN
	bStartEnabled := TRUE;
ELSE
	bStartEnabled := FALSE;
END_IF

//Handle enabling of the Stop button
IF 		eState <> Tc3_PackML_V2.E_PMLState.ePMLState_Stopped
	AND	eState <> Tc3_PackML_V2.E_PMLState.ePMLState_Clearing
	AND	eState <> Tc3_PackML_V2.E_PMLState.ePMLState_Aborted
	AND	eState <> Tc3_PackML_V2.E_PMLState.ePMLState_Aborting
	AND	eState <> Tc3_PackML_V2.E_PMLState.ePMLState_Undefined 	THEN
	bStopEnabled := TRUE;
ELSE
	bStopEnabled := FALSE;
END_IF

//Handle enabling of the Reset button
IF 		eState = Tc3_PackML_V2.E_PMLState.ePMLState_Complete
	OR	eState = Tc3_PackML_V2.E_PMLState.ePMLState_Stopped 	THEN
	bResetEnabled := TRUE;
ELSE
	bResetEnabled := FALSE;
END_IF

//Handle enabling of the Clear button
IF 		eState = Tc3_PackML_V2.E_PMLState.ePMLState_Aborted	THEN
	bClearEnabled := TRUE;
ELSE
	bClearEnabled := FALSE;
END_IF


// Handle mode changes

{warning 'add property implementation'}
PROPERTY ClearEnabled : BOOL
GET
ClearEnabled := bClearEnabled;
END_GET
SET
bClearEnabled := ClearEnabled;
END_SET
END_PROPERTY

{warning 'add property implementation'}
PROPERTY ClearPressed : BOOL
GET
ClearPressed := bClearPressed;
END_GET
SET
bClearPressed := ClearPressed;
END_SET
END_PROPERTY

PROPERTY Mode : DINT
GET
Mode := nMode;
END_GET
SET
nMode := Mode;
END_SET
END_PROPERTY

{warning 'add property implementation'}
PROPERTY ModeCommand : DINT
GET
ModeCommand := nModeCommand;
END_GET
SET
nModeCommand := ModeCommand;
END_SET
END_PROPERTY

{warning 'add property implementation'}
PROPERTY ModeCommandPulse : BOOL
GET
ModeCommandPulse := bModeCommandPulse;
END_GET
SET
bModeCommandPulse := ModeCommandPulse;
END_SET
END_PROPERTY

{warning 'add property implementation'}
PROPERTY ResetEnabled : BOOL
GET
ResetEnabled := bResetEnabled;
END_GET
SET
bResetEnabled := ResetEnabled;
END_SET
END_PROPERTY

{warning 'add property implementation'}
PROPERTY ResetPressed : BOOL
GET
bResetPressed := ResetPressed;
END_GET
SET
bResetPressed := ResetPressed;
END_SET
END_PROPERTY

{warning 'add property implementation'}
PROPERTY StartEnabled : BOOL
GET
StartEnabled := bStartEnabled;
END_GET
SET
bStartEnabled := StartEnabled;
END_SET
END_PROPERTY

{warning 'add property implementation'}
PROPERTY StartPressed : BOOL
GET
StartPressed := bStartPressed;
END_GET
SET
bStartPressed := StartPressed;
END_SET
END_PROPERTY

{warning 'add property implementation'}
PROPERTY State : Tc3_PackML_V2.E_PMLState
GET
State := eState;
END_GET
SET
eState := State;
END_SET
END_PROPERTY

{warning 'add property implementation'}
PROPERTY StateCommand : Tc3_PackML_V2.E_PMLCommand
GET
StateCommand := eStateCommand;
END_GET
SET
eStateCommand := StateCommand;
END_SET
END_PROPERTY

{warning 'add property implementation'}
PROPERTY StateCommandPulse : BOOL
GET
StateCommandPulse := bStateCommandPulse;
END_GET
SET
bStateCommandPulse := StateCommandPulse;
END_SET
END_PROPERTY

{warning 'add property implementation'}
PROPERTY StopEnabled : BOOL
GET
StopEnabled := bStopEnabled;
END_GET
SET
bStopEnabled := StopEnabled;
END_SET
END_PROPERTY

{warning 'add property implementation'}
PROPERTY StopPressed : BOOL
GET
StopPressed := bStopPressed;
END_GET
SET
bStopPressed := StopPressed;
END_SET
END_PROPERTY

END_FUNCTION_BLOCK

// ---- Base/01_PML/01_Module/03_PMLControl/FB_PackML_PushButtonControl.TcPOU
FUNCTION_BLOCK FB_PackML_PushButtonControl EXTENDS FB_PackML_ExternalControl
VAR_INPUT
END_VAR
VAR_OUTPUT
END_VAR
VAR
	bStartButton	AT %I* : BOOL;	//Tie to hardware start pushbutton
	//TODO: add other buttons
END_VAR

//TODO: implement button control

END_FUNCTION_BLOCK

// ---- Base/01_PML/01_Module/02_Events/FB_PMLStateLogger.TcPOU
FUNCTION_BLOCK FB_PMLStateLogger
VAR_IN_OUT
	a_fbPMLAlarms			: ARRAY[1..48] OF FB_TcAlarm;		//Array of alarms for Core PackML events that exist in any PackML enabled module
END_VAR
VAR_INPUT
	sModulePrefix : STRING;	//Prefix String for any
	eState	: E_PMLState;
	///Mode : DINT;
END_VAR
VAR_OUTPUT
END_VAR
VAR
	eLastState : E_PMLState := E_PMLState.ePMLState_Aborted;
END_VAR

IF eState <> eLastState THEN
	CASE eState OF
		E_PMLState.ePMLState_Starting:
			a_fbPMLAlarms[E_PMLAlarms.StateStartingEnter].Raise(0);
		E_PMLState.ePMLState_Execute:
			a_fbPMLAlarms[E_PMLAlarms.StateExecuteEnter].Raise(0);
		E_PMLState.ePMLState_Completing:
			a_fbPMLAlarms[E_PMLAlarms.StateCompletingEnter].Raise(0);
		E_PMLState.ePMLState_Complete:
			a_fbPMLAlarms[E_PMLAlarms.StateCompleteEnter].Raise(0);
		E_PMLState.ePMLState_Resetting:
			a_fbPMLAlarms[E_PMLAlarms.StateResettingEnter].Raise(0);
		E_PMLState.ePMLState_Idle:
			a_fbPMLAlarms[E_PMLAlarms.StateIdleEnter].Raise(0);
		E_PMLState.ePMLState_Holding:
			a_fbPMLAlarms[E_PMLAlarms.StateHoldingEnter].Raise(0);
		E_PMLState.ePMLState_Held:
			a_fbPMLAlarms[E_PMLAlarms.StateHeldEnter].Raise(0);
		E_PMLState.ePMLState_Unholding:
			a_fbPMLAlarms[E_PMLAlarms.StateUnholdingEnter].Raise(0);
		E_PMLState.ePMLState_Suspending:
			a_fbPMLAlarms[E_PMLAlarms.StateSuspendingEnter].Raise(0);
		E_PMLState.ePMLState_Suspended:
			a_fbPMLAlarms[E_PMLAlarms.StateSuspendedEnter].Raise(0);
		E_PMLState.ePMLState_Unsuspending:
			a_fbPMLAlarms[E_PMLAlarms.StateUnsuspendingEnter].Raise(0);
		E_PMLState.ePMLState_Stopping:
			a_fbPMLAlarms[E_PMLAlarms.StateStoppingEnter].Raise(0);
		E_PMLState.ePMLState_Stopped:
			a_fbPMLAlarms[E_PMLAlarms.StateStoppedEnter].Raise(0);
		E_PMLState.ePMLState_Aborting:
			a_fbPMLAlarms[E_PMLAlarms.StateAbortingEnter].Raise(0);
		E_PMLState.ePMLState_Aborted:
			a_fbPMLAlarms[E_PMLAlarms.StateAbortedEnter].Raise(0);
		E_PMLState.ePMLState_Clearing:
			a_fbPMLAlarms[E_PMLAlarms.StateClearingEnter].Raise(0);
		E_PMLState.ePMLState_Undefined:
			a_fbPMLAlarms[E_PMLAlarms.StateUndefinedEnter].Raise(0);

	END_CASE
	
	CASE eLastState OF
		E_PMLState.ePMLState_Starting:
			a_fbPMLAlarms[E_PMLAlarms.StateStartingEnter].Clear(0,0);
		E_PMLState.ePMLState_Execute:
			a_fbPMLAlarms[E_PMLAlarms.StateExecuteEnter].Clear(0,0);
		E_PMLState.ePMLState_Completing:
			a_fbPMLAlarms[E_PMLAlarms.StateCompletingEnter].Clear(0,0);
		E_PMLState.ePMLState_Complete:
			a_fbPMLAlarms[E_PMLAlarms.StateCompleteEnter].Clear(0,0);
		E_PMLState.ePMLState_Resetting:
			a_fbPMLAlarms[E_PMLAlarms.StateResettingEnter].Clear(0,0);
		E_PMLState.ePMLState_Idle:
			a_fbPMLAlarms[E_PMLAlarms.StateIdleEnter].Clear(0,0);
		E_PMLState.ePMLState_Holding:
			a_fbPMLAlarms[E_PMLAlarms.StateHoldingEnter].Clear(0,0);
		E_PMLState.ePMLState_Held:
			a_fbPMLAlarms[E_PMLAlarms.StateHeldEnter].Clear(0,0);
		E_PMLState.ePMLState_Unholding:
			a_fbPMLAlarms[E_PMLAlarms.StateUnholdingEnter].Clear(0,0);
		E_PMLState.ePMLState_Suspending:
			a_fbPMLAlarms[E_PMLAlarms.StateSuspendingEnter].Clear(0,0);
		E_PMLState.ePMLState_Suspended:
			a_fbPMLAlarms[E_PMLAlarms.StateSuspendedEnter].Clear(0,0);
		E_PMLState.ePMLState_Unsuspending:
			a_fbPMLAlarms[E_PMLAlarms.StateUnsuspendingEnter].Clear(0,0);
		E_PMLState.ePMLState_Stopping:
			a_fbPMLAlarms[E_PMLAlarms.StateStoppingEnter].Clear(0,0);
		E_PMLState.ePMLState_Stopped:
			a_fbPMLAlarms[E_PMLAlarms.StateStoppedEnter].Clear(0,0);
		E_PMLState.ePMLState_Aborting:
			a_fbPMLAlarms[E_PMLAlarms.StateAbortingEnter].Clear(0,0);
		E_PMLState.ePMLState_Aborted:
			a_fbPMLAlarms[E_PMLAlarms.StateAbortedEnter].Clear(0,0);
		E_PMLState.ePMLState_Clearing:
			a_fbPMLAlarms[E_PMLAlarms.StateClearingEnter].Clear(0,0);
		E_PMLState.ePMLState_Undefined:
			a_fbPMLAlarms[E_PMLAlarms.StateUndefinedEnter].Clear(0,0);

	END_CASE
	eLastState := eState;
END_IF

END_FUNCTION_BLOCK

// ---- Base/01_PML/01_Module/02_Events/FB_PMLModeLogger.TcPOU
FUNCTION_BLOCK FB_PMLModeLogger
VAR_IN_OUT
	a_fbPMLAlarms			: ARRAY[1..48] OF FB_TcAlarm;		//Array of alarms for Core PackML events that exist in any PackML enabled module
END_VAR
VAR_INPUT
	sModulePrefix : STRING;	//Prefix String for any
	///State	: E_PMLState;
	Mode : DINT;
END_VAR
VAR_OUTPUT
END_VAR
VAR
	lastMode : DINT;
END_VAR

IF Mode <> lastMode THEN
	CASE Mode OF
		E_PMLUnitMode.ePMLUnitMode_Invalid:
			a_fbPMLAlarms[E_PMLAlarms.ModeInvalidEnter].Raise(0);
		E_PMLUnitMode.ePMLUnitMode_Production:	
			a_fbPMLAlarms[E_PMLAlarms.ModeProductionEnter].Raise(0);
		E_PMLUnitMode.ePMLUnitMode_Maintenance:
			a_fbPMLAlarms[E_PMLAlarms.ModeMaintenanceEnter].Raise(0);
		E_PMLUnitMode.ePMLUnitMode_Manual:
			a_fbPMLAlarms[E_PMLAlarms.ModeManualEnter].Raise(0);
	END_CASE
	
	CASE lastMode OF
		E_PMLUnitMode.ePMLUnitMode_Invalid:
			a_fbPMLAlarms[E_PMLAlarms.ModeInvalidEnter].Clear(0,0);
		E_PMLUnitMode.ePMLUnitMode_Production:	
			a_fbPMLAlarms[E_PMLAlarms.ModeProductionEnter].Clear(0,0);
		E_PMLUnitMode.ePMLUnitMode_Maintenance:
			a_fbPMLAlarms[E_PMLAlarms.ModeMaintenanceEnter].Clear(0,0);
		E_PMLUnitMode.ePMLUnitMode_Manual:
			a_fbPMLAlarms[E_PMLAlarms.ModeManualEnter].Clear(0,0);
	END_CASE
	lastMode := Mode;
END_IF

END_FUNCTION_BLOCK

// ---- Base/03_Utilities/01_Events/F_CreateAllEventsInClass.TcPOU
FUNCTION F_CreateAllEventsInClass : BOOL
VAR_IN_OUT
	p_aAlarms : ARRAY[*] OF FB_TcAlarm;		//Array of Alarms to be defined
END_VAR
VAR_INPUT
	nClassSize : DINT;
	pInitEvent : POINTER TO TcEventEntry;	//Address of first event in Event Class (Should be the InitReferenceEvent)
	sPrefix	: STRING;	//String Prefix for the Event Message -- Usually the Module ID and Name
END_VAR
VAR
	i : DINT;
	nEventSize : DINT;
	numberOfEvents : DINT;
	pEvent	: POINTER TO TcEventEntry;
END_VAR

nEventSize := SIZEOF(pInitEvent^);
numberOfEvents := nClassSize/nEventSize;

FOR i := LOWER_BOUND(p_aAlarms,1) TO UPPER_BOUND(p_aAlarms,1) DO
	IF i > numberOfEvents THEN
		EXIT;
	ELSE
		pEvent := pInitEvent + ((i - 1) * nEventSize);
		p_aAlarms[i].CreateEx(stEventEntry := pEvent^, 0,0);
		p_aAlarms[i].ipArguments.AddString(sPrefix);
	END_IF
END_FOR

END_FUNCTION

// ---- Application/03_EquipmentModules/FB_TestEquipment.TcPOU
FUNCTION_BLOCK FB_TestEquipment EXTENDS FB_PMLModuleBase
VAR
	//Define the Sub modules here for this module.  Also set the Interfaces in the initialize method.
	//fbSubModule1				: FB_ApplicationModule_TEMPLATE;		// Sub module instantiation
	//fbSubModule2				: FB_ApplicationModule_TEMPLATE;		// Sub module instantiation
	fb_EM1_ControlModule1		: FB_TestControl;
	
	//temporary array of module base interfaces to be copied over to the base class itfPackMLBase variable
	a_itfPackMLBase_init		: ARRAY[1..MAX_NO_OF_SUBUNITS] OF ITF_PMLModuleBase := [fb_EM1_ControlModule1](*, fbSubModule2,*);

	// Other machine specific variables here
END_VAR

//*********************************************************
// Code implementation only in Execute() method for consistency with templates
//*********************************************************

// 
// Cyclic Code
METHOD CyclicLogic
VAR
	i								: UDINT;		//Generic iteration value
END_VAR
// Main loop of the parent module
SUPER^.CyclicLogic();
END_METHOD

METHOD Initialize
VAR
	i								: UDINT;		//Generic iteration value
END_VAR

// Define the interfaces to the different subunits (Must take place before SUPER^.initialize call)
FOR i := 1 TO MAX_NO_OF_SUBUNITS DO
	a_itfPackMLBase[i] := a_itfPackMLBase_init[i];
END_FOR

fb_EM1_ControlModule1.iMasterDataStructure_Adder 	:= iMasterDataStructure_Adder;
fb_EM1_ControlModule1.Enabled 						:=  TRUE;
fb_EM1_ControlModule1.ModuleName 					:=  'Test Control 1';
fb_EM1_ControlModule1.ModuleID 						:=  1;
fb_EM1_ControlModule1.AncestorIDs 					:= CONCAT(CONCAT(sAncestorIDs, DINT_TO_STRING(nModuleID)), '_');

iMasterDataStructure_Adder.AddNodeAsChildByName(fb_EM1_ControlModule1.ModuleName, sModuleName);

// Init of the parent class object (Must be called AFTER most local init code, since the sub module interface array assignments should be made here, and then operated on within the module base init
SUPER^.Initialize();
END_METHOD

END_FUNCTION_BLOCK

// ---- Application/04_ControlModules/FB_TestControl.TcPOU
FUNCTION_BLOCK FB_TestControl EXTENDS FB_PMLModuleBase
VAR
	//Define the Sub modules here for this module.  Also set the Interfaces in the initialize method.
	//fbSubModule1				: FB_ApplicationModule_TEMPLATE;		// Sub module instantiation
	//fbSubModule2				: FB_ApplicationModule_TEMPLATE;		// Sub module instantiation
	
	//temporary array of module base interfaces to be copied over to the base class itfPackMLBase variable
	a_itfPackMLBase_init		: ARRAY[1..MAX_NO_OF_SUBUNITS] OF ITF_PMLModuleBase (*:= [fbSubModule1, fbSubModule2,*);

	// Other machine specific variables here
	fbCylinder_01				: FB_Cylinder_DualSolenoid_DualSensor;
	fbCylinder_01_TestTimer_1	: TON;
	fbAxis1 : FB_Axis_Continuous_NoHoming;
END_VAR

//*********************************************************
// Code implementation only in Execute() method for consistency with templates
//*********************************************************

// 
// Cyclic Code
METHOD CyclicLogic
VAR
	i								: UDINT;		//Generic iteration value
END_VAR
// Main loop of the parent module
SUPER^.CyclicLogic();

fbAxis1.CyclicLogic();
END_METHOD

METHOD Initialize
VAR
	i								: UDINT;		//Generic iteration value
END_VAR

// Define the interfaces to the different subunits (Must take place before SUPER^.initialize call)
FOR i := 1 TO MAX_NO_OF_SUBUNITS DO
	a_itfPackMLBase[i] := a_itfPackMLBase_init[i];
END_FOR

fbCylinder_01.Enabled 			:= TRUE;
fbCylinder_01.Simulate 			:= TRUE;
fbCylinder_01.Name 				:= 'Test Cylinder 1';
fbCylinder_01_TestTimer_1.PT 	:= MAX(fbCylinder_01.ExtendTime, fbCylinder_01.RetractTime) + T#1S;

fbAxis1.Enabled		:= TRUE;
fbAxis1.Simulate	:= TRUE;
fbAxis1.Name		:= 'test Axis';


// Init of the parent class object (Must be called AFTER most local init code, since the sub module interface array assignments should be made here, and then operated on within the module base init
SUPER^.initialize();
END_METHOD

END_FUNCTION_BLOCK

// ---- Base/02_Components/03_Cylinders/03_Actuation/FB_Cylinder_DualSolenoid_DualSensor.TcPOU
FUNCTION_BLOCK FB_Cylinder_DualSolenoid_DualSensor EXTENDS FB_Cylinder_DualSensor
VAR_INPUT
END_VAR
VAR_OUTPUT
END_VAR
VAR
	bExtend_Actuator_HardwareOutput 	AT %Q* 	: BOOL;
	bRetract_Actuator_HardwareOutput 	AT %Q* 	: BOOL;
END_VAR

METHOD HardwareUpdate : BOOL
VAR_INPUT
END_VAR
SUPER^.HardwareUpdate();

bExtend_Actuator_HardwareOutput := bExtendCommand;
bRetract_Actuator_HardwareOutput := bRetractCommand;
END_METHOD

END_FUNCTION_BLOCK

// ---- Base/02_Components/03_Cylinders/02_Feedback/FB_Cylinder_DualSensor.TcPOU
FUNCTION_BLOCK FB_Cylinder_DualSensor EXTENDS FB_CylinderBase
VAR_INPUT
END_VAR
VAR_OUTPUT
END_VAR
VAR
	fbSensor_Extended							: FB_Sensor;
	fbSensor_Retracted							: FB_Sensor;
END_VAR

METHOD HardwareUpdate : BOOL
VAR_INPUT
END_VAR
fbSensor_Extended.CyclicLogic();
fbSensor_Retracted.CyclicLogic();

bExtendedFeedback:= fbSensor_Extended.Active;
bRetractedFeedback := fbSensor_Retracted.Active;
END_METHOD

END_FUNCTION_BLOCK

// ---- Base/02_Components/03_Cylinders/01_Base/FB_CylinderBase.TcPOU
FUNCTION_BLOCK ABSTRACT FB_CylinderBase EXTENDS FB_ComponentBase IMPLEMENTS ITF_CylinderBase		//Abstract (non-instantiable) base definition from which numerous varieties of Cylinders may be derived through function block extension.
VAR_INPUT
END_VAR
VAR_OUTPUT
END_VAR
VAR CONSTANT
	//Constant declarations
	CYLINDER_BASE_ALARM_COUNT	: UDINT := 16;
END_VAR
VAR
	//ITF_Cylinder internal property variables
	tExtendTime		: TIME := T#1S;		//Approximate expected time for the cylinder to complete an extension cycle
	tRetractTime 	: TIME := T#1S;		//Approximate expected time for the cylinder to complete a retraction cycle
	fTimeoutFactor	: LREAL := 1.5;		//Multiplicative factor that determines error timeout threshold based on the expected cycle time
	bExtended 		: BOOL;				//Status bit for the position of the cylinder
	bRetracted		: BOOL;				//Status bit for the position of the cylinder
	bExtending		: BOOL;				//Cylinder is currently extending
	bRetracting		: BOOL;				//Cylinder is currently retracting
	bExtendOutput	: BOOL;				//Cylinder "extend" output is currently active
	bRetractOutput	: BOOL; 			//Cylinder "retract" output is currently active

	//Alarming
	a_fbCylinderBaseAlarms : ARRAY[1..CYLINDER_BASE_ALARM_COUNT] OF FB_TcAlarm;
	
	//HMI monitoring and control structure
	stCylinderBaseHMI		: ST_CylinderBase_HMI;
	
	//Internal Variables
	fbExtensionTimeout_TON		: Tc2_Standard.TON;		//Timer for monitoring extension timeouts
	tExtensionTimeout			: TIME;					//Extension timeout threshold calculated from expected ExtendTime and TimeoutFactor
	fbRetractionTimeout_TON		: Tc2_Standard.TON;		//Timer for monitoring retraction timeouts
	tRetractionTimeout			: TIME;					//Retraction timeout threshold calculated from expected RetractTime and TimeoutFactor
	bExtendRequest				: BOOL;					//Extension request received
	bRetractRequest				: BOOL;					//Retraction request received
	bExtendCommand				: BOOL;					//Direct command to be sent to outputs
	bRetractCommand				: BOOL;					//Direct command to be sent to outputs
	bExtendedFeedback			: BOOL;					//Direct feedback value from inputs
	bRetractedFeedback			: BOOL;					//Direct feedback value from inputs
	bIncomingRequest			: BOOL;					//New external request has been made
	
	
	//Simulation variables
	fbSimExtend_TON		: Tc2_Standard.TON;
	fbSimRetract_TON	: Tc2_Standard.TON;
	bSimExtendCommand	: BOOL;
	bSimRetractCommand	: BOOL;
END_VAR

METHOD ErrorOperation : BOOL
VAR_INPUT
END_VAR
bExtendCommand := FALSE;
bRetractCommand := FALSE;
END_METHOD

METHOD Extend : BOOL
bExtendRequest := TRUE;
bRetractRequest := FALSE;
bIncomingRequest := TRUE;
END_METHOD

PROPERTY Extended : BOOL	//Status bit for the position of the cylinder
GET
Extended := bExtended;
END_GET
END_PROPERTY

PROPERTY Extending : BOOL
GET
Extending := bExtending;
END_GET
END_PROPERTY

PROPERTY ExtendOutput : BOOL
GET
ExtendOutput := bExtendOutput;
END_GET
END_PROPERTY

PROPERTY ExtendTime : TIME	//Approximate expected time for the cylinder to complete an extension cycle
GET
ExtendTime := tExtendTime;
END_GET
SET
tExtendTime := ExtendTime;
END_SET
END_PROPERTY

METHOD HMICommunication : BOOL
SUPER^.HMICommunication();		//Call the base method

//Process HMI requests
IF stCylinderBaseHMI.bIncomingHMIRequest AND NOT stCylinderBaseHMI.bHMICommandConfirmation THEN		//If a request has been issued by the HMI, and a previous request has not just finished being processed
	IF stCylinderBaseHMI.bHMIControlAvailable THEN		//If the current conditions permit HMI control (Should be determined by the extended application components)
		IF stCylinderBaseHMI.bExtendHMIRequest THEN		//Execute the active requests
			Extend();
			stCylinderBaseHMI.bHMICommandConfirmation := TRUE;	//Confirm that the request has been processed
		END_IF
		IF stCylinderBaseHMI.bRetractHMIRequest THEN
			Retract();
			stCylinderBaseHMI.bHMICommandConfirmation := TRUE;	//Confirm that the request has been processed
		END_IF
		IF stCylinderBaseHMI.bIdleHMIRequest THEN
			Idle();
			stCylinderBaseHMI.bHMICommandConfirmation := TRUE;	//Confirm that the request has been processed
		END_IF
		IF stCylinderBaseHMI.bExtendTimeHMISetRequest THEN
			ExtendTime := stCylinderBaseHMI.tExtendTimeHMISetValue;
			stCylinderBaseHMI.bHMICommandConfirmation := TRUE;	//Confirm that the request has been processed
		END_IF
		IF stCylinderBaseHMI.bRetractTimeHMISetRequest THEN
			RetractTime := stCylinderBaseHMI.tRetractTimeHMISetValue;
			stCylinderBaseHMI.bHMICommandConfirmation := TRUE;	//Confirm that the request has been processed
		END_IF
		IF stCylinderBaseHMI.bTimeoutFactorHMISetRequest THEN
			TimeoutFactor := stCylinderBaseHMI.fTimeoutFactorHMISetValue;
			stCylinderBaseHMI.bHMICommandConfirmation := TRUE;	//Confirm that the request has been processed
		END_IF
	END_IF
END_IF


//Update HMI status info
stCylinderBaseHMI.tExtendTime := tExtendTime;
stCylinderBaseHMI.tRetractTime := tRetractTime;
stCylinderBaseHMI.fTimeoutFactor := fTimeoutFactor;
stCylinderBaseHMI.bExtended := bExtended;
stCylinderBaseHMI.bExtending := bExtending;
stCylinderBaseHMI.bRetracted := bRetracted;
stCylinderBaseHMI.bRetracting := bRetracting;
stCylinderBaseHMI.bExtendCommand := bExtendCommand OR bSimExtendCommand;
stCylinderBaseHMI.bRetractCommand := bRetractCommand OR bSimRetractCommand;
END_METHOD

METHOD Idle : BOOL
bExtendRequest := FALSE;
bRetractRequest := FALSE;
bIncomingRequest := TRUE;
END_METHOD

METHOD initialize : BOOL
VAR_INPUT
END_VAR

VAR
	sTemp: STRING;
END_VAR
SUPER^.initialize();

sTemp := CONCAT(CONCAT(CONCAT('Cylinder ', ': '), sName), ' '); 	//Creates a utility string for alarms and other messaging that reads (example text) - "Module 10 - Main Casepacker" to be followed by the alarm or message info
//TODO: Rename Event Class to AxisBase
F_CreateAllEventsInClass(	p_aAlarms := a_fbCylinderBaseAlarms,
							nClassSize := SIZEOF(TC_EVENTS.CylinderBase),
							pInitEvent := ADR(TC_EVENTS.CylinderBase.InitReferenceEvent),
							sPrefix := sTemp );
END_METHOD

METHOD Monitoring : BOOL
VAR_INPUT
END_VAR
SUPER^.Monitoring();

IF NOT bError THEN
	tExtensionTimeout := LREAL_TO_TIME(TIME_TO_LREAL(tExtendTime) * fTimeoutFactor);
	tRetractionTimeout := LREAL_TO_TIME(TIME_TO_LREAL(tRetractTime) * fTimeoutFactor);
	
